//	kontroller.Din_Dout[0].kcc		:= 16#155;	// 01 - есть Целостность цепи для всех 5-ти выходов (в ЭЛПК-03-02 нет целостности выходов) 		
	K_Din_Dout_kk.kcc	:=	16#155;		// 01 - есть Целостность цепи для всех 5-ти выходов (в ЭЛПК-03-02 нет целостности выходов !!!)

//	kontroller.Din_Dout[0].value_cc	:= kontroller.Dout_[0];	//	содержимое выходных регистров		
	K_Din_Dout_kk.value_cc	:=	K_Dout;	//	содержимое выходных регистров

	// 01 - пассивное состояние			 10 - активное состояние 		
	K_Din_Dout_kk.kk.0	:=	NOT K_Dout.0;
	K_Din_Dout_kk.kk.1	:=	    K_Dout.0;
	// 01 - пассивное состояние			 10 - активное состояние 		
	K_Din_Dout_kk.kk.2	:=	NOT K_Dout.1;
	K_Din_Dout_kk.kk.3	:=	    K_Dout.1;
	// 01 - пассивное состояние			 10 - активное состояние 		
	K_Din_Dout_kk.kk.4	:=	NOT K_Dout.2;
	K_Din_Dout_kk.kk.5	:=	    K_Dout.2;
	// 01 - пассивное состояние			 10 - активное состояние 		
	K_Din_Dout_kk.kk.6	:=	NOT K_Dout.3;
	K_Din_Dout_kk.kk.7	:=	    K_Dout.3;
	// 01 - пассивное состояние			 10 - активное состояние 		
	K_Din_Dout_kk.kk.8	:=	NOT K_Dout.4;
	K_Din_Dout_kk.kk.9	:=	    K_Dout.4;

	// 01 - пассивное состояние			 10 - активное состояние 		
	K_Din_Dout_kk.kk.10	:=	NOT K_Dout.5;
	K_Din_Dout_kk.kk.11	:=	    K_Dout.5;
	// 01 - пассивное состояние			 10 - активное состояние 		
	K_Din_Dout_kk.kk.12	:=	NOT K_Dout.6;
	K_Din_Dout_kk.kk.13	:=	    K_Dout.6;
	// 01 - пассивное состояние			 10 - активное состояние 		
	K_Din_Dout_kk.kk.14	:=	NOT K_Dout.7;
	K_Din_Dout_kk.kk.15	:=	    K_Dout.7;

END_FUNCTION

// K2/std12k5/MAIN
PROGRAM MAIN
VAR

END_VAR


ELPK03_to_MLP_IN();// читать входы ЭЛПК-03-02 и передать в массивы 04

MainUP_PRG();// диагностика и OPC


///////////////////////////////////////////////////////////////////////////////////////////////////////////////////////
callExec(kontrollers);

{IF defined(imit)}
	{warning 'РЕЖИМ ИМИТАЦИИ! Входы и выходы отключены от физического источника'}
{ELSE}
execKontrollersInputs(table:=kontrollers);
{END_IF}

//SIP ();
callExec (YstTable);
callExec(imTable);
ProtectManager ();
OPC_Imit ();
algManager();
PPU_Init_ ();
Off_Q ();
{IF NOT defined(imit)}
execKontrollersOutputs(table:=kontrollers);
{END_IF}
///////////////////////////////////////////////////////////////////////////////////////////////////////////////////////

ELPK03_to_MLP_OUT(DO2_BLK:= 16#FF00, DO3_BLK:= 16#18FF);	// читать массивы 04 и передать в выходы ЭЛПК-03-02
										// с блокировкой ст байта DO_K[2] для индикации резервирования
										// с блокировкой мл байта DO_K[3] (сигналы резервирования старого) + DO_K[3].11 + DO_K[3].12 (индикация активности К1 и К2)

END_PROGRAM

// LowLevel_Algoritms/algoritms/Rassoglasovanie_dPmg
{attribute 'symbol' := 'none'}
FUNCTION_BLOCK PUBLIC Rassoglasovanie_dPmg EXTENDS BaseIM
VAR_INPUT
	di:REFERENCE TO singleSignal;
	ai:REFERENCE TO AISource;
END_VAR
VAR_OUTPUT
END_VAR
VAR
END_VAR

SUPER^();
IF	((di.q) AND (ai.value >= (ai.LA + 10))) OR ((NOT di.q) AND (ai.value <= (ai.LA - 10))) THEN
	statusSet.setBit (bitNum:=0,value:=1);
ELSE
	statusSet.setBit (bitNum:=0,value:=0);
END_IF

END_FUNCTION_BLOCK

// lowLevel_ecl/im/BaseIms/BaseIm
	{attribute 'symbol' := 'none'}
FUNCTION_BLOCK BaseIm EXTENDS BaseObject
IMPLEMENTS ObjectCommands, IImArchObject
VAR_INPUT
		{attribute 'symbol' := 'readwrite'}
	command:WORD;
END_VAR
VAR

END_VAR
VAR_OUTPUT
	{attribute 'symbol' := 'read'}
	status:DWORD;
	CommandFault:BOOL;
END_VAR
VAR
	statusSet:smartPack:=(status:=status);	
	objectTable:TableDescriptor;
	
	_command:WORD:=0;
	_haveCommand:BOOL;
	_logTwoCommands:AloneLogMessage;
	_cmd:UINT;
	_source:UINT;
	_error:UINT;
	_errorReset:TON:=(PT:=T#15S);
	_cmdReset:TON:=	(PT:=T#1S);
	_needResetCmd:BOOL;
	_opcCommandsDisabled:BOOL:=FALSE;
END_VAR

processObjectTable();

SUPER^();
_haveCommand:=FALSE;

statusSet.reset();

_errorReset(IN:=(_error<>0));

_command:=command;
command:=0;

IF _errorReset.Q THEN
	_error:=0;
	writeCommandToStatus();
END_IF

_cmdReset();
IF _needResetCmd AND _cmdReset.Q THEN
	resetCommand();
END_IF

IF hasCommand THEN
	onCommandActive(command:=_cmd);
END_IF

CommandFault:=_error<>0;

statusSet.setBit(21,_opcCommandsDisabled);

PROPERTY archName : STRING
GET
archName:=name;
END_GET
END_PROPERTY

PROPERTY archStatus : DWORD
GET
archStatus:=status;
END_GET
END_PROPERTY

METHOD PUBLIC DisableOpcControl
VAR_INPUT
END_VAR
VAR
	curObject:POINTER TO BaseObject;
	IcurIm:ObjectCommands;
END_VAR
_opcCommandsDisabled:=TRUE;

curObject:=objectTable.head;
IF curObject<>0 THEN
	REPEAT
		IF (__QUERYINTERFACE(curObject^,IcurIm)) THEN		
			IcurIm.DisableOpcControl();
		END_IF;
		curObject:=curObject^.getNext();
	UNTIL curObject=0
	END_REPEAT;
END_IF;
END_METHOD

METHOD EnableOpcControl
VAR_INPUT

END_VAR
VAR
	curObject:POINTER TO BaseObject;
	IcurIm:ObjectCommands;
END_VAR
_opcCommandsDisabled:=FALSE;

curObject:=objectTable.head;
IF curObject<>0 THEN
	REPEAT
		IF (__QUERYINTERFACE(curObject^,IcurIm)) THEN		
			IcurIm.EnableOpcControl();
		END_IF;
		curObject:=curObject^.getNext();
	UNTIL curObject=0
	END_REPEAT;
END_IF;
END_METHOD

METHOD FINAL execCommand
VAR_INPUT
END_VAR
VAR
	comUnp: SmartUnpack;
END_VAR
IF NOT _opcCommandsDisabled THEN
	IF _command<>0 THEN
		comUnp(value:=_command);	
		_source:=comUnp.getBits(13,15);
		IF _source<>0 THEN
			processCmd(cmd:=comUnp.getBits(0,2),sender:=_source,parametr:=comUnp.getBits(3,12));
		END_IF;
	END_IF;
END_IF;

ExecComands(objectTable);
END_METHOD

PROPERTY hasCommand : BOOL
GET
hasCommand:=(NOT _needResetCmd) AND (_cmd<>0);
END_GET
END_PROPERTY

PROPERTY PUBLIC opcCommandsDisabled : bool
GET
opcCommandsDisabled:=_opcCommandsDisabled;
END_GET
END_PROPERTY

METHOD PRIVATE writeCommandToStatus
VAR_INPUT
END_VAR
statusSet.setBits(23,25,_error);
statusSet.setBits(26,28,_cmd);
statusSet.setBits(29,31,_source);
END_METHOD

METHOD PROTECTED processObjectTable
VAR_INPUT
END_VAR
callExec(table:=objectTable);
END_METHOD

METHOD PROTECTED checkCmd : BOOL
VAR_INPUT
END_VAR
VAR
	
END_VAR
checkCmd:=_haveCommand;
IF _haveCommand THEN
	_logTwoCommands.write(CmpLog.LogClass.LOG_WARNING,name,'Two commands: ');
END_IF
_haveCommand:=TRUE;
END_METHOD

METHOD PROTECTED resetCommand
VAR_INPUT
END_VAR
IF _cmdReset.Q THEN
	_cmd:=0;
	_source:=0;
	writeCommandToStatus();
	_cmdReset(IN:=FALSE);
	_needResetCmd:=FALSE;
ELSE
	_needResetCmd:=TRUE;
END_IF;
END_METHOD

METHOD PROTECTED errorCommand
VAR_INPUT
END_VAR
_error:=_cmd;
resetCommand();
END_METHOD

//Метод вызывается каждый такт пересчета пока идет выполенение команды.
METHOD PROTECTED onCommandActive
VAR_INPUT
	command:WORD;
END_VAR
errorCommand();
END_METHOD

METHOD PROTECTED processCmd;
VAR_INPUT
	cmd:UINT;
	sender:UINT;
	parametr:UINT;
END_VAR
END_METHOD

METHOD PROTECTED setCmd
VAR_INPUT
	nCmd:uint;
END_VAR
checkCmd();
_cmd:=nCmd;
_error:=0;

_cmdReset(in:=FALSE);
_cmdReset.IN:=TRUE;	
	
_needResetCmd:=FALSE;
writeCommandToStatus();
END_METHOD

METHOD PUBLIC sendCommand
VAR_INPUT
	source:cmdSources;
	parametr:UINT;
	cmd:UINT;
END_VAR
_command:= SHL(source AND 16#7,13) OR SHL(parametr AND 16#3FF ,3) OR (cmd AND 16#3);
execCommand();
END_METHOD

METHOD PUBLIC writeImStatus
VAR_INPUT
END_VAR
END_METHOD

METHOD PUBLIC CommandFail : bool
VAR_INPUT
END_VAR
CommandFail:=_error<>0;
END_METHOD

END_FUNCTION_BLOCK

// lowLevel_ecl/Common/smartPack/smartPack
	{attribute 'symbol' := 'none'}
	{attribute 'reflection'}
FUNCTION_BLOCK smartPack//Упаковывает биты в двойное слово. 
(*Выдает ошибку в журнал если полсе reset() записывались одни и теже биты.
*)
VAR_INPUT	
	status:REFERENCE TO DWORD;//указатель на двойное слово
END_VAR
VAR_OUTPUT
END_VAR
VAR
	settedBits:DWORD;
	bitsAlredySetted:AloneLogMessage;
	bitsOutOfRenge:AloneLogMessage;
	{attribute 'instance-path'} 
	{attribute 'noinit'} 
	name: STRING; 
END_VAR
VAR CONSTANT

END_VAR

METHOD PUBLIC reset //сброс контроля перезаписи
VAR_INPUT
END_VAR
settedBits:=0;
END_METHOD

METHOD setBit 
//установить 1 бит
VAR_INPUT
	bitNum:WORD;// номер бита (с 0)
	value:BOOL;//Значение бита
END_VAR
setBits(bitNum,bitNum,bool_to_word(value));
END_METHOD

METHOD PUBLIC setBits //Устанавливает последовательность бит
VAR_INPUT
	start:WORD;//номер первого бита(с 0) 
	end:WORD;//номер последнего бита(с 0)
	value:DWORD;//значение. Записывается start-end+1 младших бит.
END_VAR
VAR
	statusMask:DWORD;
	bitsCount:WORD;
END_VAR
IF (start<0) OR (start>31) OR (end<0) OR (end>31) OR (start>end) THEN
	bitsOutOfRenge.write(CmpLog.LogClass.LOG_ERROR,name,'Nums out of range: ');	
	RETURN;
END_IF

bitsCount:=end-start+1;
statusMask:=SHL(SHL(1,bitsCount)-1,start);
IF (settedBits AND statusMask)<>0 THEN
	bitsAlredySetted.write(CmpLog.LogClass.LOG_ERROR,name,'Conflict bits: ');
END_IF
settedBits:=settedBits OR statusMask;
status:=(status AND NOT statusMask) OR (SHL(value,start) AND statusMask);
END_METHOD

END_FUNCTION_BLOCK

// lowLevel_ecl/Common/smartPack/SmartUnpack
{attribute 'symbol' := 'none'}
FUNCTION_BLOCK SmartUnpack//Распаковывает слово
VAR_INPUT
	value:WORD; //Значение
END_VAR
VAR_OUTPUT
END_VAR
VAR
END_VAR

METHOD getBit : BOOL
VAR_INPUT
	start:WORD;
END_VAR
getBit:= getBits(start,start)<>0;
END_METHOD

METHOD getBits : Word
VAR_INPUT
	start:WORD;
	end: WORD;
END_VAR
VAR
	statusMask:WORD;
	bitsCount:WORD;
END_VAR
bitsCount:=end-start+1;
statusMask:=SHL(SHL(1,bitsCount)-1,start);
getBits:=SHR(value AND statusMask,start);
END_METHOD

END_FUNCTION_BLOCK

// lowLevel_ecl/im/BaseIms/singleSignal
{attribute 'symbol' := 'none'}
FUNCTION_BLOCK singleSignal EXTENDS BaseIm
VAR_INPUT
	signal:REFERENCE TO ReliableBit;
END_VAR
VAR_OUTPUT
	Q:BOOL;
	reliability:BOOL;
END_VAR
VAR
END_VAR

SUPER^();
IF __ISVALIDREF(signal) THEN
	Q:=checkArg(signal);
	reliability:=signal.reliability;
END_IF

METHOD PUBLIC writeImStatus
VAR_INPUT
END_VAR
SUPER^.writeImStatus();
statusSet.setBit(0,Q);
END_METHOD

END_FUNCTION_BLOCK

// lowLevel_ecl/Common/functions/checkArg
FUNCTION checkArg : BOOL
VAR_INPUT
	chBit:REFERENCE TO ReliableBit;
END_VAR
VAR
END_VAR

checkArg:=FALSE;
IF __ISVALIDREF(chBit) THEN
	IF chBit.reliability THEN
		checkArg:=chBit.value;
	END_IF
END_IF

END_FUNCTION

// lowLevel_ecl/kontroller/baseSources/ReliableBit
	{attribute 'symbol' := 'none'}
FUNCTION_BLOCK ReliableBit
VAR_INPUT
END_VAR
VAR_OUTPUT
	value:BOOL;//Значение	
	reliability:BOOL;//достоверный
END_VAR
VAR
	
END_VAR

PROPERTY PUBLIC ReliableFalse : Bool
GET
ReliableFalse:= (NOT value) AND reliability;
END_GET
END_PROPERTY

PROPERTY PUBLIC ReliableTrue : Bool
GET
ReliableTrue:=value AND reliability;
END_GET
END_PROPERTY

METHOD setReliability
VAR_INPUT
	rel:BOOL;
END_VAR
reliability:=rel;
END_METHOD

METHOD PUBLIC setValue
VAR_INPUT
	val: BOOL;
END_VAR
value:=val;
END_METHOD

END_FUNCTION_BLOCK

// lowLevel_ecl/kontroller/baseSources/AISource
	{attribute 'symbol' := 'none'}
FUNCTION_BLOCK AISource EXTENDS BaseIm
IMPLEMENTS ISource, IAnalogArchObject, IAiSource
VAR_INPUT
	addr:WORD;
	
	dLL:REAL:=RNaN(); 
	dHL:REAL:=RNaN(); 
	dLA:REAL:=RNaN();
	dHA:REAL:=RNaN();
	dLW:REAL:=RNaN();
	dHW:REAL:=RNaN();  
	dmaxChangeSpeed:REAL:=RNaN();  
END_VAR
VAR_OUTPUT
		{attribute 'symbol' := 'readwrite'}
	value:REAL;

	interval:statusAi;
	
	remont	:	BOOL	;	//	bit-0 вывод канала в ремонт  1-есть, 0 –нет				
	{attribute 'symbol' := 'read'} 
	LL	:	REAL	:=RNaN();	//	Нижняя граница физического диапазона	Для преобразования из 4-20 мА и отображения в SCADA.
	{attribute 'symbol' := 'read'} 
	HL	:	REAL	:=RNaN();	//	Верхняя граница физического диапазона	Для преобразования из 4-20 мА и отображения в SCADA.
	{attribute 'symbol' := 'read'} 
	HA	:	REAL	:=RNaN();	//	Верхняя аварийная граница	Уставка срабатывания аварийного останова по повышению параметра
	{attribute 'symbol' := 'read'} 
	HW	:	REAL	:=RNaN();	//	Верхняя предупредительная граница	Уставка срабатывания предупредительной сигнализации по повышению параметра
	{attribute 'symbol' := 'read'} 
	LW	:	REAL	:=RNaN();	//	Нижняя предупредительная граница	Уставка срабатывания предупредительной сигнализации по понижению параметра
	{attribute 'symbol' := 'read'} 
	LA	:	REAL	:=RNaN();	//	Верхняя аварийная граница	Уставка срабатывания аварийного останова по понижению параметра
	{attribute 'symbol' := 'read'} 
	histeresis	:	REAL	;	//	Гистерезис.( % от физической шкалы) Уставка устранения дребезга по предупредительной сигнализации	Для устранения частого срабатывания предупредительной сигнализации при колебания около границы	
	//_de	:	REAL	;	//	Уставка рассогласования от аппаратных границ	Разница тока для формирования неисправности канала по выходу за диапазон измерения.
	{attribute 'symbol' := 'read'} 
	aperturFilter	:	REAL	;	//	Уставка апертурного фильтра	При применении апертурного фильтра, фильтрация малых изменений сигнала
	{attribute 'symbol' := 'read'} 
	pikFiler	:	REAL	;	//	Уставка пикового фильтра	При применении пикового фильтра, фильтрация пиков, случайных бросков сигнала
	{attribute 'symbol' := 'read'} 
	exponentialFilter	:	REAL	:=RNaN();	//	Уставка экпоненциального фильтра	При применении экспоненциального фильтра.
	{attribute 'symbol' := 'read'}
	rassoglasovanie	:	REAL	;	//	Уставка рассогласования от аппаратных границ. В процентах от диапазона.
	{attribute 'symbol' := 'read'}	
	maxChangeSpeed:REAL; //Максимальная скорость изменения сигнала 1/сек
	{attribute 'symbol' := 'read'} 
	ChangeSpeed:REAL;//Скорость изменения.
END_VAR
VAR
	{attribute 'symbol' := 'readwrite'}
	newLL:REAL;  // новые границы
	{attribute 'symbol' := 'readwrite'}
	newHL:REAL;  // новые границы
	{attribute 'symbol' := 'readwrite'}
	newLA:REAL;  // новые границы
	{attribute 'symbol' := 'readwrite'}
	newHA:REAL;  // новые границы
	{attribute 'symbol' := 'readwrite'}
	newLW:REAL;  // новые границы
	{attribute 'symbol' := 'readwrite'}
	newHW:REAL;  // новые границы		

	_imit:BOOL;  
	_notReliable:BOOL;
	_disabledAlarms:BYTE;
	
	_lastValue:REAL:=RNaN();
	_LastValueTimer:TON:=(PT:=T#1S);
	_normalTrig:R_TRIG;
END_VAR

VAR CONSTANT
	cmd_SetUstavki:WORD:=1;
	cmd_SetRemont:WORD:=2;
	cmd_ResetRemont:WORD:=3;
	cmd_kvitNotReliable:WORD:=4;
END_VAR
VAR_TEMP
	srcInterval:statusAi;
END_VAR

SUPER^();

IF NOT imit THEN
	value:=getData(o_interval=>srcInterval);
	
	value:=apFilter(value,_lastValue);
	value:=exponential(value,_lastValue);
ELSE
	srcInterval:=statusAi.normal;
END_IF;

IF NOT notReliable THEN
	IF srcInterval=statusAi.normal THEN
		interval:=CalkLimits();
	ELSE
		interval:=srcInterval;
	END_IF;
ELSE
	interval:=statusAi.NOTRELIABLE;
END_IF	

IF remont THEN
	interval:=statusAi.NOTDEFINED;
END_IF


_normalTrig(CLK:=interval>=statusAi.normal);

IF (NOT FPU.IsRealNaN(_lastValue)) AND (NOT _normalTrig.Q) THEN
	_LastValueTimer();
	IF (value<>_lastValue) OR _LastValueTimer.Q THEN
		IF (_LastValueTimer.ET>T#0MS) THEN
			ChangeSpeed:=(value-_lastValue)/(TIME_TO_REAL(_LastValueTimer.ET)/1000);
		END_IF
		_LastValueTimer(IN:=FALSE);
		_LastValueTimer(IN:=TRUE);
	END_IF
END_IF

_lastValue:=value;

IF (NOT FPU.IsRealNaN(maxChangeSpeed)) AND (maxChangeSpeed>0) THEN
	IF (interval>=statusAi.normal) THEN		
		IF ABS(ChangeSpeed)>maxChangeSpeed THEN
			 notReliable:=TRUE;
		END_IF
	END_IF
END_IF

PROPERTY aiInterval : statusAi
GET
aiInterval:=interval;
END_GET
END_PROPERTY

PROPERTY aiRemont : BOOL
GET
aiRemont:=remont;
END_GET
END_PROPERTY

PROPERTY aiValue : REAL
GET
aiValue:=value;
END_GET
END_PROPERTY

METHOD PRIVATE apFilter: REAL
VAR_INPUT
	currentValue:REAL;
	lastValue:REAL;
END_VAR
VAR
	ap:REAL;
END_VAR
IF NOT FPU.IsRealNaN(aperturFilter) THEN
	ap:=aperturFilter*0.01*(Hl-Ll);
	IF rABS(currentValue-lastValue)>ap THEN
		apFilter:=currentValue;
	ELSE
		apFilter:=lastValue;
	END_IF
ELSE
	apFilter:=currentValue;
END_IF
END_METHOD

PROPERTY archName : STRING
GET
END_GET
END_PROPERTY

PROPERTY archSrcValue : REAL
GET
END_GET
END_PROPERTY

PROPERTY archStatus : DWORD
GET
END_GET
END_PROPERTY

PROPERTY archValue : REAL
GET
archValue:=value;
END_GET
END_PROPERTY

METHOD PROTECTED CalkLimits:statusAi
VAR_INPUT

END_VAR
VAR
	h:REAL:=0;
	mismatch:REAL:=0;
END_VAR
CalkLimits:=statusAi.NOTDEFINED;

IF NOT (FPU.IsRealNaN(ll) OR FPU.IsRealNaN(Hl))THEN
	h := histeresis* 0.01 * (Hl-Ll);
	mismatch:=rassoglasovanie* 0.01 * (Hl-Ll);
	
	IF ( value < LL-mismatch)   THEN
		CalkLimits:=statusAi.LL;
		RETURN;
	END_IF  
	IF  (value > Hl+mismatch) THEN
		CalkLimits:=statusAi.HL;
		RETURN;
	END_IF
END_IF

IF (NOT FPU.IsRealNaN(la)) AND ((disabledAlarms AND AnalogAlarms.LA)=0) THEN
	IF (value  < La) OR ((interval=statusAi.LA)  AND ( (value -h) < La))  THEN 
		CalkLimits:=statusAi.LA;
		RETURN;
	END_IF
END_IF 

IF NOT FPU.IsRealNaN(Ha) AND ((disabledAlarms AND AnalogAlarms.HA)=0)THEN
	IF (value > Ha) OR ((interval=statusAi.HA)  AND ( (value +h) > HA))  THEN 
		CalkLimits:=statusAi.HA;
		RETURN;
	END_IF
END_IF

IF NOT FPU.IsRealNaN(LW) AND ((disabledAlarms AND AnalogAlarms.LW)=0) THEN
	IF (value < LW) OR ((interval=statusAi.LW)  AND ( (value -h) < Lw))   THEN 
		CalkLimits:=statusAi.LW;
		RETURN;
	END_IF
END_IF

IF NOT FPU.IsRealNaN(HW) AND ((disabledAlarms AND AnalogAlarms.HW)=0)THEN
	IF (value  > HW)  OR ((interval=statusAi.HW)  AND ( (value +h) > Hw))   THEN 
		CalkLimits:=statusAi.HW;
		RETURN;
	END_IF
END_IF

CalkLimits:=statusAi.normal;
END_METHOD

{attribute 'symbol' := 'none'}
PROPERTY PUBLIC disabledAlarms : BYTE
GET
disabledAlarms:=_disabledAlarms;
END_GET
SET
_disabledAlarms:=disabledAlarms;
END_SET
END_PROPERTY

METHOD PRIVATE exponential : Real
VAR_INPUT
	currentValue:REAL;
	lastValue:REAL;
END_VAR
IF (NOT FPU.IsRealNaN(exponentialFilter)) AND (exponentialFilter<>0) AND (NOT FPU.IsRealNaN(lastValue)) THEN
	exponential:=exponentialFilter*currentValue+(1-exponentialFilter)*lastValue;
ELSE
	exponential:=currentValue;
END_IF
END_METHOD

METHOD PROTECTED GetData : Real
VAR_INPUT
END_VAR
VAR_OUTPUT
	o_interval:statusAi;
END_VAR
END_METHOD

{attribute 'symbol' := 'none'}
PROPERTY imit : BOOL
GET
imit:=_imit;
END_GET
SET
_imit:=imit;
END_SET
END_PROPERTY

METHOD kvitNotReliable
VAR_INPUT
END_VAR
setCmd(nCmd:=cmd_kvitNotReliable);

_notReliable:=FALSE;

resetCommand();
END_METHOD

{attribute 'symbol' := 'none'}
PROPERTY PUBLIC notReliable : bool
GET
notReliable:=_notReliable;
END_GET
SET
IF notReliable THEN
	_notReliable:=notReliable;
	interval:=statusAi.NOTRELIABLE;
END_IF
END_SET
END_PROPERTY

METHOD PROTECTED processCmd;
VAR_INPUT
	cmd:UINT;
	sender:UINT;
	parametr:UINT;
END_VAR
CASE cmd OF
	cmd_SetUstavki:setUstavki(nLL:=newLL,nLA:=newLA, nLW:=newLW, nHW:=newHW, nHa:=newHA,nHl:=newHL,flags:= parametr);
	cmd_SetRemont:setRemont();
	cmd_ResetRemont:resetRemont();
	cmd_kvitNotReliable:kvitNotReliable();
END_CASE
END_METHOD

METHOD PROTECTED readPersistent
VAR_INPUT
END_VAR
Ll:=FPU.StrToReal(readValue());
la:=FPU.StrToReal(readValue());
lw:=FPU.StrToReal(readValue());
hw:=FPU.StrToReal(readValue());
ha:=FPU.StrToReal(readValue());
Hl:=FPU.StrToReal(readValue());
remont:=STRING_TO_BOOL(readValue());
histeresis:=FPU.StrToReal(readValue());
aperturFilter:=FPU.StrToReal(readValue());
pikFiler:=FPU.StrToReal(readValue());
exponentialFilter:=FPU.StrToReal(readValue());
rassoglasovanie:=FPU.StrToReal(readValue());
maxChangeSpeed:=FPU.StrToReal(readValue());
END_METHOD

METHOD resetRemont
VAR_INPUT
END_VAR
setCmd(nCmd:=cmd_ResetRemont);

remont:=FALSE;

SaveToFile();

resetCommand();
END_METHOD

METHOD PROTECTED setDefaultPersistent:BOOL
VAR_INPUT
END_VAR
LL:=dLL;
LA:=dLA;
LW:=dLW;
HW:=dHW;
Ha:=dHA;
Hl:=dHL;
maxChangeSpeed:=dmaxChangeSpeed;
setDefaultPersistent:=TRUE;
END_METHOD

METHOD setRemont
VAR_INPUT
END_VAR
setCmd(nCmd:=cmd_SetRemont);

remont:=TRUE;

SaveToFile();

resetCommand();
END_METHOD

METHOD setUstavki
VAR_INPUT
	nLL:REAL;
	nHl:REAL;
	nLA:REAL;
	nHa:REAL;
	nLW:REAL;
	nHW:REAL;
	flags:WORD:=16#FF;
END_VAR
setCmd(nCmd:=cmd_SetUstavki);

IF (flags AND AnalogLimitFlags.LL)<>0 THEN
	LL:=nLL;
END_IF
IF (flags AND AnalogLimitFlags.HL)<>0 THEN
	Hl:=nHl;
END_IF
IF (flags AND AnalogLimitFlags.LA)<>0 THEN
	LA:=nlA;
END_IF
IF (flags AND AnalogLimitFlags.HA)<>0 THEN
	Ha:=nha;
END_IF
IF (flags AND AnalogLimitFlags.LW)<>0 THEN
	LW:=nlW;
END_IF
IF (flags AND AnalogLimitFlags.HW)<>0 THEN
	HW:=nhw;
END_IF

SaveToFile();

resetCommand();
END_METHOD

METHOD PUBLIC writeImStatus
VAR_INPUT
END_VAR
VAR
	cInteval:statusAi;
END_VAR
SUPER^.writeImStatus();
statusSet.setBits(0,3,interval);
statusSet.setBit(4,remont);
statusSet.setBit(5,interval<statusAi.normal);
statusSet.setBits(6,9,_disabledAlarms);
END_METHOD

METHOD PROTECTED writePersistent
VAR_INPUT
END_VAR
writeValue(value:=FPU.RealToStr(Ll),comment:='LL');
writeValue(value:=FPU.RealToStr(la),comment:='LA');
writeValue(value:=FPU.RealToStr(lw),comment:='LW');
writeValue(value:=FPU.RealToStr(hw),comment:='HW');
writeValue(value:=FPU.RealToStr(ha),comment:='HA');
writeValue(value:=FPU.RealToStr(Hl),comment:='HL');
writeValue(value:=BOOL_TO_STRING(remont),comment:='Ремонт');
writeValue(value:=FPU.RealToStr(histeresis),comment:='Гистерезис');
writeValue(value:=FPU.RealToStr(aperturFilter),comment:='Апертурный фильтр');
writeValue(value:=FPU.RealToStr(pikFiler),comment:='Пиковый фильтр');
writeValue(value:=FPU.RealToStr(exponentialFilter),comment:='Экспоненциальный фильтр');
writeValue(value:=FPU.RealToStr(rassoglasovanie),comment:='Рассогласование');
writeValue(value:=FPU.RealToStr(maxChangeSpeed),comment:='Максимальная скорость изменения');
END_METHOD

END_FUNCTION_BLOCK

// lowLevel_ecl/kontroller/baseSources/IAiSource
INTERFACE IAiSource

PROPERTY aiInterval : statusAi
GET
END_GET
END_PROPERTY

PROPERTY aiRemont : BOOL
GET
END_GET
END_PROPERTY

PROPERTY aiValue : real
GET
END_GET
END_PROPERTY

END_INTERFACE

// lowLevel_ecl/Common/functions/RNaN
FUNCTION RNaN : real
VAR_INPUT
END_VAR
VAR
END_VAR

RNaN:=FPU.GetRealSpecialVal(fpu.ESpecial_FP_Value.NaN);

END_FUNCTION

// lowLevel_ecl/Common/functions/rABS
FUNCTION rABS : real
VAR_INPUT
	inp:REAL;
END_VAR
VAR
END_VAR

IF inp<0.0 THEN
	rABS:=-inp;
ELSE
	rABS:=inp;
END_IF

END_FUNCTION

// K1/std12k5/modbus/tstModbus
	{attribute 'symbol' := 'none'}
FUNCTION_BLOCK tstModbus EXTENDS MbKontroller
VAR_INPUT
END_VAR
VAR_OUTPUT
	di_1:DiSourceMb(table:=ADR(inputTable)):=(addr:=0);
	ai_1:AiSourceMb(table:=ADR(inputTable)):=(addr:=1,reliability:=di_1.bits[1]);
	ao_1:AoProxiMb(table:=ADR(outputTable)):=(addr:=5, source:=ai_1);
END_VAR
VAR
END_VAR

SUPER^();

METHOD PROTECTED ProcessInputs
VAR_INPUT
END_VAR
IF di_1.trigs[5].Qp THEN
	//команда
END_IF
END_METHOD

METHOD PROTECTED ProcessOutputs
VAR_INPUT
END_VAR
setOutputValue(addr:=5,1);
setOutputFloat(addr:=6,1.5);
END_METHOD

END_FUNCTION_BLOCK

// K2/std12k5/modbus/tstModbus
	{attribute 'symbol' := 'none'}
FUNCTION_BLOCK tstModbus EXTENDS MbKontroller
VAR_INPUT
END_VAR
VAR_OUTPUT
	di_1:DiSourceMb(table:=ADR(inputTable)):=(addr:=0);
	ai_1:AiSourceMb(table:=ADR(inputTable)):=(addr:=1,reliability:=di_1.bits[1]);
	ao_1:AoProxiMb(table:=ADR(outputTable)):=(addr:=5, source:=ai_1);
END_VAR
VAR
END_VAR

SUPER^();

METHOD PROTECTED ProcessInputs
VAR_INPUT
END_VAR
IF di_1.trigs[5].Qp THEN
	//команда
END_IF
END_METHOD

METHOD PROTECTED ProcessOutputs
VAR_INPUT
END_VAR
setOutputValue(addr:=5,1);
setOutputFloat(addr:=6,1.5);
END_METHOD

END_FUNCTION_BLOCK

// lowLevel_ecl/kontroller/modbus/MbKontroller
{attribute 'symbol' := 'none'}
FUNCTION_BLOCK MbKontroller EXTENDS baseKontroller
VAR_INPUT
	MbRole:MbKontrollerRole;
	slaveError:REFERENCE TO BOOL;
	slaveRestart:REFERENCE TO BOOL;
	restartDelay:TIME:=T#20S;
	restartDuration:TIME:=T#30S;
	AiWordOrder:MbAiWordOrder:=MbAiWordOrder.AiWordOrder12;
END_VAR
VAR_OUTPUT
	{attribute 'symbol' := 'read'}
	noLink:BOOL;
END_VAR
VAR
	input:ARRAY [1..500] OF WORD;
	holding:ARRAY [1..500] OF WORD;
	
	_init:BOOL;
	
	restartTimer:TON;
	noLinkTimer:TOF;
END_VAR

SUPER^();
IF NOT _init THEN
	setSourcesProp(table:=inputTable);
	setSourcesProp(table:=outputTable);
	_init:=TRUE;
END_IF
IF NOT imit THEN
	IF (__ISVALIDREF(slaveError)) THEN
		noLinkTimer(IN:=slaveError,PT:=restartDuration,Q=>noLink);
		IF (__ISVALIDREF(slaveRestart)) THEN
			restartTimer(IN:=slaveError AND (NOT slaveRestart),PT:=restartDelay,Q=>slaveRestart);
		END_IF
	END_IF
ELSE
	noLink:=FALSE;
END_IF

METHOD PUBLIC callInputTable
VAR_INPUT
END_VAR
SUPER^.callInputTable();
ProcessInputs();
END_METHOD

METHOD callOutputTable
VAR_INPUT
END_VAR
ProcessOutputs();
SUPER^.callOutputTable();
END_METHOD

METHOD PUBLIC getInputFloat : REAL
VAR_INPUT
	addr:WORD;
END_VAR
VAR
	rawValue:FloatAsWords;
END_VAR
CASE AiWordOrder OF
	MbAiWordOrder.AiWordOrder12:
		rawValue.wValue[0]:=getInputValue(addr:=addr);
		rawValue.wValue[1]:=getInputValue(addr:=addr+1);	
	MbAiWordOrder.AiWordOrder21:
		rawValue.wValue[0]:=getInputValue(addr:=addr+1);
		rawValue.wValue[1]:=getInputValue(addr:=addr);
END_CASE

getInputFloat:=rawValue.fValue;
END_METHOD

METHOD PUBLIC getInputValue : WORD
VAR_INPUT
	addr:WORD;
END_VAR
CASE MbRole OF
	MbKontrollerRole.MK_MASTER:
		getInputValue:=input[addr];
	MbKontrollerRole.MK_SLAVE:
		getInputValue:=holding[addr];
END_CASE
END_METHOD

METHOD PROTECTED ProcessInputs
VAR_INPUT
END_VAR
END_METHOD

METHOD PROTECTED ProcessOutputs
VAR_INPUT
END_VAR
END_METHOD

METHOD PUBLIC setOutputByte
VAR_INPUT
	addr:WORD;
	value:BYTE;
	usedByte:UsedByteMBSource;
END_VAR
VAR
	rawValue:FloatAsWords;
	
END_VAR


CASE MbRole OF
	MbKontrollerRole.MK_MASTER: 	
	rawValue.wValue[0]:=	holding[addr]; // сохраняем 
			IF usedByte=UsedByteMBSource.HB THEN 
				rawValue.bValue[1]:=	value;
			ELSE
				rawValue.bValue[0]:=	value;
			END_IF
		holding[addr]:=rawValue.wValue[0]; //кормим слово

	MbKontrollerRole.MK_SLAVE: 	
		rawValue.wValue[0]:=	input[addr]; // сохраняем 
			IF usedByte=UsedByteMBSource.HB THEN 
				rawValue.bValue[1]:=	value;
			ELSE
				rawValue.bValue[0]:=	value;
			END_IF
		input[addr]:=rawValue.wValue[0]; //кормим слово
END_CASE
END_METHOD

METHOD PUBLIC setOutputFloat
VAR_INPUT
	addr:WORD;
	value:REAL;
END_VAR
VAR
	rawValue:FloatAsWords;
END_VAR
rawValue.fValue:=value;
CASE AiWordOrder OF
	MbAiWordOrder.AiWordOrder12:
		setOutputValue(addr:=addr,value:=rawValue.wValue[0]);
		setOutputValue(addr:=addr+1,value:=rawValue.wValue[1]);	
	MbAiWordOrder.AiWordOrder21:
		setOutputValue(addr:=addr+1,value:=rawValue.wValue[0]);
		setOutputValue(addr:=addr,value:=rawValue.wValue[1]);	
END_CASE
END_METHOD

METHOD PUBLIC setOutputValue
VAR_INPUT
	addr:WORD;
	value:WORD;
END_VAR
CASE MbRole OF
	MbKontrollerRole.MK_MASTER:
		holding[addr]:=value;
	MbKontrollerRole.MK_SLAVE:
		input[addr]:=value;
END_CASE
END_METHOD

METHOD PRIVATE setSourcesProp
VAR_INPUT
	CONSTANT table:TableDescriptor;
END_VAR
VAR
	curObject:POINTER TO BaseObject;
	curSource:IMbSource;
END_VAR
curObject:=table.head;
IF curObject=0 THEN
	RETURN;
END_IF
REPEAT
	IF (__QUERYINTERFACE(curObject^,curSource)) THEN		
		curSource.setKontroller(THIS^);
	END_IF;
	curObject:=curObject^.getNext();
	UNTIL curObject=0
END_REPEAT
END_METHOD

END_FUNCTION_BLOCK

// lowLevel_ecl/kontroller/modbus/Sources/IMbSource
INTERFACE IMbSource EXTENDS __SYSTEM.IQueryInterface

METHOD setKontroller
VAR_INPUT
	nKontroller:REFERENCE TO MbKontroller;
END_VAR
END_METHOD

END_INTERFACE

// lowLevel_ecl/kontroller/modbus/Sources/DiSourceMb
{attribute 'symbol' := 'none'}
FUNCTION_BLOCK DiSourceMb EXTENDS DISource
IMPLEMENTS IMbSource;
VAR_INPUT
	
END_VAR
VAR_OUTPUT
	Trigs:array [0..15] OF RP_trig;
END_VAR
VAR
	mbKontr:REFERENCE TO MbKontroller;
	bitNumber:INT;
	I:INT;
END_VAR

SUPER^();

FOR I:=0 TO 15 DO
	IF bits[I].reliability THEN
  		Trigs[i](in:= bits[I].value);
	END_IF
END_FOR

METHOD PROTECTED getData : word
VAR_INPUT
END_VAR
VAR_OUTPUT
	reliability:WORD;
END_VAR
getData:=mbKontr.getInputValue(addr:=addr);
IF NOT mbKontr.noLink THEN
	reliability:=16#FFFF;
ELSE
	reliability:=16#0000;	
END_IF
END_METHOD

METHOD setKontroller
VAR_INPUT
	nKontroller	: REFERENCE TO MbKontroller;
END_VAR
mbKontr REF=nKontroller;
END_METHOD

END_FUNCTION_BLOCK

// lowLevel_ecl/kontroller/baseSources/DISource
	{attribute 'symbol' := 'none'}
FUNCTION_BLOCK DISource EXTENDS BaseObject
IMPLEMENTS ISource, IDiscretArchObject
VAR_INPUT
	addr:WORD;
END_VAR
VAR_OUTPUT
		bits:ARRAY [0..15] OF InversableReliableBit;
		{attribute 'symbol' := 'readwrite'}
		value:WORD;
		{attribute 'symbol' := 'readwrite'}
		reliability:WORD;
END_VAR
VAR
	_imit:BOOL;  
END_VAR
VAR_TEMP
	bitNumber:INT;
END_VAR

SUPER^();
IF NOT imit THEN
	value:=getData(reliability=>reliability);
END_IF;

FOR bitNumber:=0 TO 15 DO
	bits[bitNumber].setReliability(UINT_TO_BOOL(SHR (reliability, bitNumber) AND 16#1));
	IF bits[bitNumber].reliability THEN
		bits[bitNumber].setValue(UINT_TO_BOOL(SHR (value, bitNumber) AND 16#1));
	END_IF;
END_FOR

PROPERTY archName : STRING
GET
archName:=name;
END_GET
END_PROPERTY

PROPERTY archReliability : WORD
GET
archReliability:=reliability;
END_GET
END_PROPERTY

PROPERTY archValue : WORD
GET
archValue:=value;
END_GET
END_PROPERTY

METHOD PROTECTED getData : word
VAR_INPUT
END_VAR
VAR_OUTPUT
	reliability:WORD;
END_VAR
END_METHOD

{attribute 'symbol' := 'none'}
PROPERTY imit : BOOL
GET
imit:=_imit;
END_GET
SET
_imit:=imit;
END_SET
END_PROPERTY

END_FUNCTION_BLOCK

// lowLevel_ecl/kontroller/baseSources/InversableReliableBit
	{attribute 'symbol' := 'none'}
FUNCTION_BLOCK InversableReliableBit EXTENDS ReliableBit
VAR_INPUT
END_VAR
VAR_OUTPUT

END_VAR
VAR
	_inversed:ReliableBit;
END_VAR

{attribute 'symbol' := 'none'}
PROPERTY inverse : REFERENCE TO ReliableBit;
GET
inverse ref=_inversed;
END_GET
END_PROPERTY

METHOD setReliability
VAR_INPUT
	rel:BOOL;
END_VAR
SUPER^.setReliability(rel);
_inversed.setReliability(rel);
END_METHOD

METHOD PUBLIC setValue
VAR_INPUT
	val: BOOL;
END_VAR
SUPER^.setValue(val);
_inversed.setValue(NOT val);
END_METHOD

END_FUNCTION_BLOCK

// lowLevel_ecl/kontroller/modbus/Sources/AiSourceMb
{attribute 'symbol' := 'none'}
FUNCTION_BLOCK AiSourceMb EXTENDS AISource
IMPLEMENTS IMbSource;
VAR_INPUT
	k:REAL:=1;
	b:REAL:=0;
	reliability:REFERENCE TO ReliableBit;
	extInterval:REFERENCE TO DISource;
END_VAR
VAR_OUTPUT
END_VAR
VAR
	mbKontr:REFERENCE TO MbKontroller;
	source:AnalogRecalc;
END_VAR

SUPER^();

METHOD PROTECTED GetData : Real
VAR_INPUT
END_VAR
VAR_OUTPUT
	o_interval:statusAi;
END_VAR
VAR
	intervalUnp:SmartUnpack;
END_VAR
source.input:=mbKontr.getInputFloat(addr:=addr);
source.k:=k;
source.b:=b;
source.h:=histeresis;
source.ap:=aperturFilter;
source.dp:=pikFiler;
source.ds:=exponentialFilter;
source.de:=rassoglasovanie;
source();

GetData:=source.value;

IF (mbKontr.noLink) AND NOT _imit THEN
	o_interval:=statusAi.NOTDEFINED;
ELSE
	IF (__ISVALIDREF(extInterval)) THEN
		intervalUnp.value:=extInterval.value;
		o_interval:=WORD_TO_BYTE(intervalUnp.getBits(0,3));
	ELSE
		IF __ISVALIDREF(reliability) THEN
			IF reliability.reliability AND reliability.value THEN
				o_interval:=statusAi.normal;
			ELSE
				o_interval:=statusAi.NOTDEFINED;
			END_IF
		ELSE
			o_interval:=statusAi.normal;	
		END_IF
	END_IF
END_IF
END_METHOD

METHOD setKontroller
VAR_INPUT
	nKontroller	: REFERENCE TO MbKontroller;
END_VAR
mbKontr REF=nKontroller;
END_METHOD

END_FUNCTION_BLOCK

// lowLevel_ecl/Common/fb/AnalogRecalc
	{attribute 'symbol' := 'none'}
FUNCTION_BLOCK AnalogRecalc
VAR_INPUT		
	k:REAL;
	b:REAL;
	input:REAL;//входное значение
	
	h	:	REAL	;	//	Гистерезис.( % от физической шкалы) Уставка устранения дребезга по предупредительной сигнализации	Для устранения частого срабатывания предупредительной сигнализации при колебания около границы
	ap	:	REAL	;	//	Уставка апертурного фильтра	При применении апертурного фильтра, фильтрация малых изменений сигнала 
	dp	:	REAL	;	//	Уставка пикового фильтра	При применении пикового фильтра, фильтрация пиков, случайных бросков сигнала 
	ds	:	REAL	;	//	Уставка экпоненциального фильтра	При применении экспоненциального фильтра.

	de	:	REAL	;	//	Уставка рассогласования от аппаратных границ	Разница тока для формирования неисправности канала по выходу за диапазон измерения.
END_VAR
VAR_OUTPUT
	value:REAL;
END_VAR
VAR
END_VAR
VAR_TEMP
END_VAR

	value := k*input +b;

END_FUNCTION_BLOCK

// lowLevel_ecl/kontroller/modbus/Sources/AoProxiMb
{attribute 'symbol' := 'none'}
FUNCTION_BLOCK PUBLIC AoProxiMb EXTENDS AOSource
IMPLEMENTS IMbSource;
VAR_INPUT
	k:REAL:=1;
	b:REAL:=0;
	Source:REFERENCE TO AISource;
END_VAR
VAR_OUTPUT
END_VAR
VAR
	mbKontr:REFERENCE TO MbKontroller;
END_VAR

SUPER^();

METHOD setKontroller
VAR_INPUT
	nKontroller: REFERENCE TO MbKontroller;
END_VAR
mbKontr REF=nKontroller;
END_METHOD

METHOD PROTECTED writeData
VAR_INPUT
	val:REAL;
END_VAR
VAR
	rawValue:FloatAsWords;	
END_VAR
IF __ISVALIDREF(Source) THEN
	rawValue.fValue:=Source.value;
	mbKontr.setOutputValue(addr:=addr+2,value:=Source.interval);
ELSE
	rawValue.fValue:=k*val+b;	
END_IF

mbKontr.setOutputFloat(addr:=addr,value:=rawValue.fValue);
END_METHOD

END_FUNCTION_BLOCK

// lowLevel_ecl/kontroller/baseSources/AOSource
	{attribute 'symbol' := 'none'}
FUNCTION_BLOCK AOSource EXTENDS BaseIm
IMPLEMENTS ISource, IAnalogArchObject
VAR_INPUT
	addr:WORD;
	
		{attribute 'symbol' := 'readwrite'}
	newLL	:	REAL	;	//	Нижняя граница физического диапазона	Для преобразования из 4-20 мА и отображения в SCADA.
		{attribute 'symbol' := 'readwrite'}
	newHL	:	REAL	;	//	Верхняя граница физического диапазона	Для преобразования из 4-20 мА и отображения в SCADA.
	
	dLL:REAL:=RNaN(); 
	dHL:REAL:=RNaN(); 
END_VAR
VAR_OUTPUT
		{attribute 'symbol' := 'read'}
	Value:REAL;
	
		{attribute 'symbol' := 'read'}
	LL	:	REAL	;	//	Нижняя граница физического диапазона	Для преобразования из 4-20 мА и отображения в SCADA.
	{attribute 'symbol' := 'read'}
	HL	:	REAL	;	//	Верхняя граница физического диапазона	Для преобразования из 4-20 мА и отображения в SCADA.	
END_VAR
VAR
		{attribute 'symbol' := 'readwrite'}
	newValue:REAL;

	_imit:BOOL;  
END_VAR

VAR CONSTANT
	cmd_ChangeValue:WORD:=1;
	cmd_ChangeLimits:WORD:=2;
END_VAR

SUPER^();
IF NOT imit THEN
	writeData(val:=Value);
END_IF;
resetCommand();

PROPERTY archSrcValue : REAL
GET
END_GET
END_PROPERTY

PROPERTY archValue : REAL
GET
archValue:=value;
END_GET
END_PROPERTY

METHOD PRIVATE cmdSetValue
VAR_INPUT
	nValue:REAL;
END_VAR
setCmd(cmd_ChangeValue);
setValue(nValue:=nValue);
END_METHOD

{attribute 'symbol' := 'none'}
PROPERTY imit : BOOL
GET
imit:=_imit;
END_GET
SET
_imit:=imit;
END_SET
END_PROPERTY

METHOD PROTECTED processCmd;
VAR_INPUT
	cmd:UINT;
	sender:UINT;
	parametr:UINT;
END_VAR
CASE cmd OF
	cmd_ChangeValue:cmdSetValue(newValue);
	cmd_ChangeLimits:setLimits();
END_CASE
END_METHOD

METHOD PROTECTED readPersistent
VAR_INPUT
END_VAR
Ll:=FPU.StrToReal(readValue());
Hl:=FPU.StrToReal(readValue());
END_METHOD

METHOD PROTECTED setDefaultPersistent:BOOL
VAR_INPUT
END_VAR
LL:=dLL;
Hl:=dHL;
setDefaultPersistent:=TRUE;
END_METHOD

METHOD setLimits
VAR_INPUT
END_VAR
setCmd(nCmd:=cmd_ChangeLimits);
Ll:=newLl;
Hl:=newHl;

SaveToFile();
END_METHOD

METHOD PUBLIC setValue
VAR_INPUT
	nValue:REAL;
END_VAR
IF ((FPU.IsRealNaN(Ll))OR(nValue>=Ll)) AND ((FPU.IsRealNaN(Hl))OR(nValue<=Hl) ) THEN
	Value:=nValue;
END_IF
END_METHOD

METHOD PROTECTED writeData
VAR_INPUT
	val:REAL;
END_VAR
END_METHOD

METHOD PROTECTED writePersistent
VAR_INPUT
END_VAR
writeValue(value:=FPU.RealToStr(LL),comment:='LL');
writeValue(value:=FPU.RealToStr(Hl),comment:='HL');
END_METHOD

END_FUNCTION_BLOCK

// LowLevel_Algoritms/algoritms/AiProtectionDual
	{attribute 'symbol' := 'none'}
FUNCTION_BLOCK AiProtectionDual EXTENDS BaseProtection
VAR_INPUT
	ai1:REFERENCE TO AISource;
	ai2:REFERENCE TO AISource;
	controlLimit:statusAi;
	control_Normal:statusAi;
	{attribute 'symbol' := 'read'}
	delay:TimeParametr(table:=ADR(objectTable));	
END_VAR
VAR_OUTPUT
END_VAR
VAR
	timer:TON;
END_VAR

SUPER^();
IF __ISVALIDREF(ai1) AND __ISVALIDREF(ai2) THEN
	timer(IN:=(	((ai1.interval=controlLimit) AND (ai2.interval=controlLimit)) OR 
				((ai1.interval=controlLimit) AND (ai2.interval < control_Normal)) OR 
				((ai2.interval=controlLimit) AND (ai1.interval < control_Normal))),PT:=delay.Value);
	IF timer.Q THEN
		signaling:=TRUE; 
	ELSE
		signaling:=FALSE;
	END_IF
END_IF

METHOD PUBLIC reset
VAR_INPUT
END_VAR
SUPER^.reset();
timer(in:=FALSE);
signaling:=FALSE;
END_METHOD

END_FUNCTION_BLOCK

// lowLevel_ecl/algoritms/BaseProtection
	{attribute 'symbol' := 'none'}
FUNCTION_BLOCK BaseProtection EXTENDS BaseAlgoritm IMPLEMENTS IProtection
VAR_INPUT
END_VAR
VAR_OUTPUT
	
END_VAR
VAR
	_remont:BOOL;
	_signaling:BOOL;
	_check:BOOL;
	
	_signalingTp:TOF:=(PT:=T#1s);
END_VAR
VAR CONSTANT
	cmd_check:UINT:=3;
	cmd_setRemont:UINT:=4;
	cmd_resetRemont:UINT:=5;
END_VAR

SUPER^();

METHOD PUBLIC check
VAR_INPUT
END_VAR
setCmd(nCmd:=cmd_check);
_check:=TRUE;
resetCommand();
END_METHOD

METHOD PROTECTED processCmd;
VAR_INPUT
	cmd:UINT;
	sender:UINT;
	parametr:UINT;
END_VAR
SUPER^.processCmd(cmd,sender,parametr);
CASE cmd OF
	cmd_SetRemont:setRemont();
	cmd_ResetRemont:resetRemont();
END_CASE
END_METHOD

METHOD PROTECTED readPersistent
VAR_INPUT
END_VAR
SUPER^.readPersistent();
_remont:=STRING_TO_BOOL(readValue());
IF remont THEN
	reset();
END_IF
END_METHOD

PROPERTY PUBLIC remont : BOOL
GET
remont:=_remont;
END_GET
SET
PRIVATE
VAR
END_VAR
IF (NOT remont) AND (_signaling) THEN
	signaling:=FALSE;
	THIS^();
END_IF
IF ((NOT _signaling) OR (remont)) THEN
	_remont:=remont;
END_IF
END_SET
END_PROPERTY

METHOD reset
VAR_INPUT
END_VAR
VAR
	curObject:POINTER TO BaseObject;
	curPhase:IAlgoritmPhase;
END_VAR
signaling:=FALSE;
_check:=FALSE;
SUPER^.reset();
END_METHOD

METHOD PUBLIC resetRemont
VAR_INPUT
END_VAR
setCmd(nCmd:=cmd_resetRemont);
remont:=FALSE;
IF (NOT remont) THEN
	resetCommand();
ELSE
	errorCommand();
END_IF
END_METHOD

METHOD PUBLIC run
VAR_INPUT
END_VAR
IF (NOT remont) THEN
	SUPER^.run();
ELSE
	setCmd(nCmd:=cmdRun);
	errorCommand();	
END_IF
END_METHOD

METHOD PUBLIC setRemont
VAR_INPUT
END_VAR
setCmd(nCmd:=cmd_setRemont);
remont:=TRUE;
resetCommand();
END_METHOD

PROPERTY PUBLIC signaling : BOOL
GET
IF (NOT remont) AND (NOT _check) THEN
	signaling:=_signaling;
ELSE
	signaling:=FALSE;
END_IF
END_GET
SET
PROTECTED 
VAR
END_VAR
_signaling:=signaling;
IF NOT remont THEN
	_signalingTp(in:=_signaling);
ELSE
	_signalingTp(in:=FALSE);
END_IF
END_SET
END_PROPERTY

METHOD PUBLIC writeImStatus
VAR_INPUT
END_VAR
SUPER^.writeImStatus();
_signalingTp();
statusSet.setBit(3,_signalingTp.Q);
statusSet.setBit(5,_check);
statusSet.setBit(6,remont);
END_METHOD

METHOD PROTECTED writePersistent
VAR_INPUT
END_VAR
SUPER^.writePersistent();
writeValue(value:=BOOL_TO_STRING(_remont),comment:='Ремонт');
END_METHOD

END_FUNCTION_BLOCK

// lowLevel_ecl/algoritms/BaseAlgoritm
	{attribute 'symbol' := 'none'}
FUNCTION_BLOCK BaseAlgoritm EXTENDS BaseIm
IMPLEMENTS AlgoritmInterface
VAR_INPUT
	runOnStart:BOOL:=FALSE;
END_VAR
VAR_OUTPUT
END_VAR
VAR
	_runing:BOOL;
	_ended:BOOL;
	_CanRun: BOOL:=TRUE;
	_hasError:BOOL;
END_VAR
VAR CONSTANT
	cmdRun:WORD:=1;
	cmdReset:WORD:=2;
END_VAR

//Вызов Super^() сдесь не нужен

PROPERTY autoRun : bool
GET
autoRun:=runOnStart;
END_GET
END_PROPERTY

METHOD PUBLIC FINAL callBase
VAR_INPUT
END_VAR
VAR

END_VAR
SUPER^();
writeImStatus();
END_METHOD

PROPERTY CanRun : BOOL
GET
CanRun:=_CanRun;
END_GET
SET
_CanRun:=CanRun;
END_SET
END_PROPERTY

METHOD PROTECTED end
VAR_INPUT
END_VAR
_ended:=true;
END_METHOD

METHOD PUBLIC getTable :POINTER TO TableDescriptor
VAR_INPUT
END_VAR
getTable:=adr(objectTable);
END_METHOD

PROPERTY PUBLIC hasError : bool
GET
hasError:=_hasError;
END_GET
SET
PROTECTED 
VAR
END_VAR
_hasError:=hasError;
END_SET
END_PROPERTY

PROPERTY PUBLIC isEnded : bool
GET
isEnded:=_ended;
END_GET
END_PROPERTY

PROPERTY isRuning : BOOL
GET
isRuning:=_runing;
END_GET
END_PROPERTY

METHOD PROTECTED onInit
VAR_INPUT
END_VAR
VAR
	curObject:POINTER TO BaseObject;
	IcurAlg:AlgoritmInterface;
END_VAR
SUPER^.onInit();

curObject:=objectTable.head;
IF curObject<>0 THEN
	REPEAT
		IF (__QUERYINTERFACE(curObject^,IcurAlg)) THEN	
			IcurAlg.callBase();
			IcurAlg.reset();
			IF IcurAlg.autoRun THEN
				IcurAlg.run();
			END_IF
		END_IF;
		curObject:=curObject^.getNext();
	UNTIL curObject=0
	END_REPEAT;
END_IF;
END_METHOD

METHOD PROTECTED processCmd;
VAR_INPUT
	cmd:UINT;
	sender:UINT;
	parametr:UINT;
END_VAR
CASE cmd OF
	cmdRun:
		run();
	cmdReset:
		reset();
END_CASE
END_METHOD

METHOD PROTECTED processObjectTable
VAR_INPUT
END_VAR
VAR
		curObject:POINTER TO BaseObject;
		IcurAlg:AlgoritmInterface;
END_VAR
curObject:=objectTable.head;
IF curObject<>0 THEN
	REPEAT
		IF (__QUERYINTERFACE(curObject^,IcurAlg)) THEN
			IcurAlg.callBase();	
			IF IcurAlg.isRuning THEN	
				curObject^();
			END_IF;			
		ELSE
			callObject(curObject);			
		END_IF;
	
		curObject:=curObject^.getNext();
	UNTIL curObject=0
	END_REPEAT;
END_IF;
END_METHOD

METHOD reset
VAR_INPUT
END_VAR
VAR
	curObject:POINTER TO BaseObject;
	curPhase:IAlgoritmPhase;
END_VAR
setCmd(cmdReset);
end();
_runing:=FALSE;
_ended:=FALSE;
resetCommand();
END_METHOD

METHOD run
VAR_INPUT
END_VAR
VAR
	curObject:POINTER TO BaseObject;
	curPhase:IAlgoritmPhase;
END_VAR
setCmd(cmdRun);
IF (CanRun) THEN
	_runing:=TRUE;
	resetCommand();
ELSE
	errorCommand();
END_IF
END_METHOD

METHOD PUBLIC writeImStatus
VAR_INPUT
END_VAR
statusSet.setBit(0,isRuning);
statusSet.setBit(1,_ended);
statusSet.setBit(2,_canRun);
statusSet.setBit(4,hasError);
END_METHOD

END_FUNCTION_BLOCK

// lowLevel_ecl/algoritms/AlgoritmInterface
INTERFACE AlgoritmInterface EXTENDS __SYSTEM.IQueryInterface

PROPERTY autoRun : bool
GET
END_GET
END_PROPERTY

METHOD PUBLIC callBase
VAR_INPUT
END_VAR
END_METHOD

PROPERTY CanRun : bool
GET
END_GET
SET
END_SET
END_PROPERTY

PROPERTY isRuning : bool
GET
END_GET
END_PROPERTY

METHOD reset
VAR_INPUT
END_VAR
END_METHOD

METHOD run
VAR_INPUT
END_VAR
END_METHOD

END_INTERFACE

// lowLevel_ecl/algoritms/phases/IAlgoritmPhase
INTERFACE IAlgoritmPhase EXTENDS __SYSTEM.IQueryInterface

PROPERTY error : Bool
GET
END_GET
END_PROPERTY

METHOD getPhaseNum : UINT
VAR_INPUT
END_VAR
END_METHOD

METHOD reset : Bool
VAR_INPUT
END_VAR
END_METHOD

METHOD run
VAR_INPUT
END_VAR
END_METHOD

METHOD setBlockIm
VAR_INPUT
	algRuning:BOOL;
END_VAR
END_METHOD

PROPERTY start : Bool
GET
END_GET
END_PROPERTY

PROPERTY top : Bool
GET
END_GET
END_PROPERTY

END_INTERFACE

// lowLevel_ecl/algoritms/IProtection
INTERFACE IProtection

METHOD PUBLIC check
VAR_INPUT
END_VAR
END_METHOD

PROPERTY PUBLIC remont : BOOL
GET
END_GET
END_PROPERTY

PROPERTY PUBLIC signaling : BOOL
GET
END_GET
END_PROPERTY

END_INTERFACE

// lowLevel_ecl/Common/parameters/TimeParametr
	{attribute 'symbol' := 'none'}
FUNCTION_BLOCK TimeParametr EXTENDS BaseIm
VAR_INPUT
		{attribute 'symbol' := 'readwrite'}
	newValue:TIME;	
END_VAR
VAR_OUTPUT
		{attribute 'symbol' := 'read'}
	Value:TIME;
END_VAR
VAR
	
END_VAR
VAR CONSTANT
	cmd_ChangeValue:WORD:=1;
END_VAR


SUPER^();

resetCommand();

METHOD PROTECTED processCmd;
VAR_INPUT
	cmd:UINT;
	sender:UINT;
	parametr:UINT;
END_VAR
CASE cmd OF
	cmd_ChangeValue:setValue(newValue);
END_CASE
END_METHOD

METHOD PROTECTED readPersistent
VAR_INPUT
END_VAR
Value:=STRING_TO_TIME(readValue());
END_METHOD

METHOD PUBLIC setValue
VAR_INPUT
	nValue:TIME;
END_VAR
setCmd(cmd_ChangeValue);
Value:=nValue;

SaveToFile();
END_METHOD

METHOD PROTECTED writePersistent
VAR_INPUT
END_VAR
writeValue(value:=TIME_TO_STRING(Value),comment:='value');
END_METHOD

END_FUNCTION_BLOCK

// K1/std12k5/AlgoritmsManager
	{attribute 'symbol' := 'none'}
FUNCTION_BLOCK AlgoritmsManager EXTENDS BaseAlgoritmsManager
VAR_INPUT
END_VAR
VAR_OUTPUT
	{attribute 'symbol' := 'read'}
	mode:ModeGpa;
	reg_V:BOOL;
END_VAR
VAR
	AoTrig:F_TRIG;
END_VAR

SUPER^();

METHOD PROTECTED onStart
VAR_INPUT
END_VAR
algoritms.opcComands.CanRun:=TRUE;
algoritms.opcComands.run();
///*ТЕМПЕРАТУРЫ*///////
(*Температуры т.1 - т.10*) 
		protections.p_TOpornogoPodshipnikaEDT_1.run();
		protections.p_TOpornoYpornogoPodshipnikaEDT_2.run();
		protections.p_TOpornoYpornogoPodshipnikaKolesaRedEDT_3.run();
		protections.p_TOpornoYpornogoPodshipnikaKolesaRedHT_4.run();
		protections.p_TOpornogoPodshipnikaShesterniReduktoraT_5.run();
		protections.p_TOpornogoPodshipnikaReduktoraHT_6.run();
		protections.p_TOpornoYpornogoPodshipnikaNagnetateljaT_7.run();
																										
		protections.p_TOpornoYpornogoPodshipnikaSvobodnogoKoncaNT_8.run();
		protections.p_TYpornogoPodshipnikaRavKolodokHT_9.run();
		protections.p_TYpornogoPodshipnikaNerabKolodokHT_10.run();
		protections.p_TgazaNaVyhodeH.run();
		
	(*Давления*)
		
		protections.p_OsSdvigNagnetatelja_Plus.run();
		protections.p_OsSdvigNagnetatelja_Minus.run();
		
	
	(*Дискретные сигналы *)
		
		
		protections.p_AO_PRU.run();
		protections.p_AO_fromSHU.run();
					
		algoritms.Synch_Rejim_.CanRun:=TRUE;
		algoritms.Synch_Rejim_.run ();
		
im.mv.DisableOpcControl ();
im.kran1.DisableOpcControl ();
im.kran2.DisableOpcControl ();
im.kran3.DisableOpcControl ();
im.kran3b.DisableOpcControl ();
im.kran4.DisableOpcControl ();
im.kran5.DisableOpcControl ();
END_METHOD

METHOD PROTECTED onInit
VAR_INPUT
END_VAR
VAR
	curObject:POINTER TO BaseObject;
	IcurAlg:AlgoritmInterface;
END_VAR
SUPER^.onInit();
setMode(nMode:=ModeGpa.MODE_STOP);
END_METHOD

METHOD PUBLIC setMode
VAR_INPUT
	nMode:ModeGpa;
END_VAR
IF 	nMode<>mode THEN
	mode:=nMode;
	CASE 	mode OF
	mode_stop:	resetAndDisable(alg:=algoritms.Auto_Avom_);
		resetAndDisable(alg:=algoritms.autoNu_1);
		resetAndDisable(alg:=algoritms.autoNu_2);
		resetAndDisable(alg:=algoritms.autoPns);
		resetAndDisable(alg:=algoritms.AUto_Ten_);
		resetAndDisable(alg:=algoritms.PNS_ON_MV_);
		resetAndDisable(alg:=algoritms.no);
		resetAndDisable(alg:=algoritms.ao);
		resetAndDisable(alg:=algoritms.Pms);
		resetAndDisable(alg:=algoritms.dPmg);
		resetAndDisable(alg:=algoritms.F1_1);
		resetAndDisable(alg:=algoritms.F1_2);
		resetAndDisable(alg:=algoritms.F2_Ch);
		resetAndDisable(alg:=algoritms.F2_R);
		resetAndDisable(alg:=algoritms.F3);
		resetAndDisable(alg:=algoritms.F4);
		resetAndDisable(alg:=algoritms.Kr6_Move);
		resetAndDisable(alg:=algoritms.AutoPNS_Start);
		resetAndDisable(alg:=algoritms.R_AutoAVom);
		resetAndDisable(alg:=algoritms.S_AutoAVOM);
		resetAndDisable(alg:=algoritms.S_Vibr);
		resetAndDisable(alg:=algoritms.S_dPmg);
		resetAndDisable(alg:=algoritms.S_I);
		resetAndDisable(alg:=algoritms.S_K);
		resetAndDisable(alg:=algoritms.S_Pms);
		resetAndDisable(alg:=algoritms.S_V);
		resetAndDisable(alg:=algoritms.S_AP);
		resetAndDisable(alg:=algoritms.S_PP);
		resetAndDisable(alg:=algoritms.Test_IM);
		algoritms.Opres.CanRun:=TRUE;
		algoritms.ppu.CanRun:=TRUE;
		resetAndDisable(alg:=algoritms.R_AutoTEN);
		//algoritms.R_AutoTEN.CanRun:=TRUE;
		algoritms.S_AutoTEN.CanRun:=TRUE;
		algoritms.S_Test_IM.CanRun:=TRUE;
		resetAndDisable(alg:=algoritms.R_TestIM);
		algoritms.S_NO.CanRun:=TRUE;
		algoritms.S_AO.CanRun:=TRUE;
		algmanager.reg_V:=FALSE;
		algoritms.Start_Test_P.CanRun:=TRUE;
		resetAndDisable(alg:=algoritms.Test_P);
		algoritms.Test_P.DisableOpcControl();
		
		////////////*АЛГОРИТМЫ РАБОТАЮЩИЕ В РЕЖИМЕ АВТОМАТИЧЕСКИЙ Реакторный  ПУСК*/////////////////////////////////
MODE_PUSKAP_R:
	resetAndDisable(alg:=algoritms.Auto_Avom_);
	resetAndDisable(alg:=algoritms.autoNu_1);
	resetAndDisable(alg:=algoritms.autoNu_2);
	resetAndDisable(alg:=algoritms.autoPns);
	resetAndDisable(alg:=algoritms.AUto_Ten_);
	resetAndDisable(alg:=algoritms.PNS_ON_MV_);
	resetAndDisable(alg:=algoritms.no);
	resetAndDisable(alg:=algoritms.ao);
	resetAndDisable(alg:=algoritms.Opres);
	resetAndDisable(alg:=algoritms.Pms);
	resetAndDisable(alg:=algoritms.dPmg);
	algoritms.ppu.CanRun:=TRUE;
	algoritms.ppu.run();
	resetAndDisable(alg:=algoritms.F1_2);
	resetAndDisable(alg:=algoritms.F2_Ch);
	resetAndDisable(alg:=algoritms.F2_R);
	resetAndDisable(alg:=algoritms.F3);
	resetAndDisable(alg:=algoritms.F4);
	resetAndDisable(alg:=algoritms.Kr6_Move);
	resetAndDisable(alg:=algoritms.AutoPNS_Start);
	resetAndDisable(alg:=algoritms.R_AutoAVom);
	resetAndDisable(alg:=algoritms.R_AutoTEN);
	resetAndDisable(alg:=algoritms.R_TestIM);
	resetAndDisable(alg:=algoritms.S_AutoAVOM);
	resetAndDisable(alg:=algoritms.S_AutoTEN);
	resetAndDisable(alg:=algoritms.S_Test_IM);
	resetAndDisable(alg:=algoritms.S_Vibr);
	resetAndDisable(alg:=algoritms.S_dPmg);
	resetAndDisable(alg:=algoritms.S_I);
	resetAndDisable(alg:=algoritms.S_K);
	resetAndDisable(alg:=algoritms.S_Pms);
	resetAndDisable(alg:=algoritms.S_V);
	resetAndDisable(alg:=algoritms.S_PP);
	algoritms.S_AP.CanRun:=FALSE;
	algoritms.S_NO.CanRun:=TRUE;
	algoritms.S_AO.CanRun:=TRUE;
	resetAndDisable(alg:=algoritms.Test_IM);
	resetAndDisable(alg:=algoritms.Start_Test_P);
	resetAndDisable(alg:=algoritms.Test_P);
MODE_PUSKAP_Ch:
	resetAndDisable(alg:=algoritms.Auto_Avom_);
	resetAndDisable(alg:=algoritms.autoNu_1);
	resetAndDisable(alg:=algoritms.autoNu_2);
	resetAndDisable(alg:=algoritms.autoPns);
	resetAndDisable(alg:=algoritms.AUto_Ten_);
	resetAndDisable(alg:=algoritms.PNS_ON_MV_);
	resetAndDisable(alg:=algoritms.no);
	resetAndDisable(alg:=algoritms.ao);
	resetAndDisable(alg:=algoritms.Opres);
	resetAndDisable(alg:=algoritms.Pms);
	resetAndDisable(alg:=algoritms.dPmg);
	algoritms.ppu.CanRun:=TRUE;
	algoritms.ppu.run();
	resetAndDisable(alg:=algoritms.F1_2);
	resetAndDisable(alg:=algoritms.F2_Ch);
	resetAndDisable(alg:=algoritms.F2_R);
	resetAndDisable(alg:=algoritms.F3);
	resetAndDisable(alg:=algoritms.F4);
	resetAndDisable(alg:=algoritms.Kr6_Move);
	resetAndDisable(alg:=algoritms.AutoPNS_Start);
	resetAndDisable(alg:=algoritms.R_AutoAVom);
	resetAndDisable(alg:=algoritms.R_AutoTEN);
	resetAndDisable(alg:=algoritms.R_TestIM);
	resetAndDisable(alg:=algoritms.S_AutoAVOM);
	resetAndDisable(alg:=algoritms.S_AutoTEN);
	resetAndDisable(alg:=algoritms.S_Test_IM);
	resetAndDisable(alg:=algoritms.S_Vibr);
	resetAndDisable(alg:=algoritms.S_dPmg);
	resetAndDisable(alg:=algoritms.S_I);
	resetAndDisable(alg:=algoritms.S_K);
	resetAndDisable(alg:=algoritms.S_Pms);
	resetAndDisable(alg:=algoritms.S_V);
	resetAndDisable(alg:=algoritms.S_PP);
	algoritms.S_AP.CanRun:=FALSE;
	algoritms.S_NO.CanRun:=TRUE;
	algoritms.S_AO.CanRun:=TRUE;
	resetAndDisable(alg:=algoritms.Test_IM);
	resetAndDisable(alg:=algoritms.Start_Test_P);
	resetAndDisable(alg:=algoritms.Test_P);
MODE_PUSKPP_R:
	resetAndDisable(alg:=algoritms.Auto_Avom_);
	resetAndDisable(alg:=algoritms.autoNu_1);
	resetAndDisable(alg:=algoritms.autoNu_2);
	resetAndDisable(alg:=algoritms.autoPns);
	resetAndDisable(alg:=algoritms.AUto_Ten_);
	resetAndDisable(alg:=algoritms.PNS_ON_MV_);
	resetAndDisable(alg:=algoritms.no);
	resetAndDisable(alg:=algoritms.ao);
	resetAndDisable(alg:=algoritms.Opres);
	resetAndDisable(alg:=algoritms.Pms);
	resetAndDisable(alg:=algoritms.dPmg);
	algoritms.ppu.CanRun:=TRUE;
	algoritms.ppu.run();
	resetAndDisable(alg:=algoritms.F1_2);
	resetAndDisable(alg:=algoritms.F2_Ch);
	resetAndDisable(alg:=algoritms.F2_R);
	resetAndDisable(alg:=algoritms.F3);
	resetAndDisable(alg:=algoritms.F4);
	resetAndDisable(alg:=algoritms.Kr6_Move);
	resetAndDisable(alg:=algoritms.AutoPNS_Start);
	resetAndDisable(alg:=algoritms.R_AutoAVom);
	resetAndDisable(alg:=algoritms.R_AutoTEN);
	resetAndDisable(alg:=algoritms.R_TestIM);
	resetAndDisable(alg:=algoritms.S_AutoAVOM);
	resetAndDisable(alg:=algoritms.S_AutoTEN);
	resetAndDisable(alg:=algoritms.S_Test_IM);
	resetAndDisable(alg:=algoritms.S_Vibr);
	resetAndDisable(alg:=algoritms.S_dPmg);
	resetAndDisable(alg:=algoritms.S_I);
	resetAndDisable(alg:=algoritms.S_K);
	resetAndDisable(alg:=algoritms.S_Pms);
	resetAndDisable(alg:=algoritms.S_V);
	resetAndDisable(alg:=algoritms.S_AP);
	algoritms.S_PP.CanRun:=FALSE;
	algoritms.S_NO.CanRun:=TRUE;
	algoritms.S_AO.CanRun:=TRUE;
	resetAndDisable(alg:=algoritms.Test_IM);
	resetAndDisable(alg:=algoritms.Start_Test_P);
	resetAndDisable(alg:=algoritms.Test_P);
MODE_PUSKPP_Ch:
	resetAndDisable(alg:=algoritms.Auto_Avom_);
	resetAndDisable(alg:=algoritms.autoNu_1);
	resetAndDisable(alg:=algoritms.autoNu_2);
	resetAndDisable(alg:=algoritms.autoPns);
	resetAndDisable(alg:=algoritms.AUto_Ten_);
	resetAndDisable(alg:=algoritms.PNS_ON_MV_);
	resetAndDisable(alg:=algoritms.no);
	resetAndDisable(alg:=algoritms.ao);
	resetAndDisable(alg:=algoritms.Opres);
	resetAndDisable(alg:=algoritms.Pms);
	resetAndDisable(alg:=algoritms.dPmg);
	algoritms.ppu.CanRun:=TRUE;
	algoritms.ppu.run();
	resetAndDisable(alg:=algoritms.F1_2);
	resetAndDisable(alg:=algoritms.F2_Ch);
	resetAndDisable(alg:=algoritms.F2_R);
	resetAndDisable(alg:=algoritms.F3);
	resetAndDisable(alg:=algoritms.F4);
	resetAndDisable(alg:=algoritms.Kr6_Move);
	resetAndDisable(alg:=algoritms.AutoPNS_Start);
	resetAndDisable(alg:=algoritms.R_AutoAVom);
	resetAndDisable(alg:=algoritms.R_AutoTEN);
	resetAndDisable(alg:=algoritms.R_TestIM);
	resetAndDisable(alg:=algoritms.S_AutoAVOM);
	resetAndDisable(alg:=algoritms.S_AutoTEN);
	resetAndDisable(alg:=algoritms.S_Test_IM);
	resetAndDisable(alg:=algoritms.S_Vibr);
	resetAndDisable(alg:=algoritms.S_dPmg);
	resetAndDisable(alg:=algoritms.S_I);
	resetAndDisable(alg:=algoritms.S_K);
	resetAndDisable(alg:=algoritms.S_Pms);
	resetAndDisable(alg:=algoritms.S_V);
	resetAndDisable(alg:=algoritms.S_AP);
	algoritms.S_PP.CanRun:=FALSE;
	algoritms.S_NO.CanRun:=TRUE;
	algoritms.S_AO.CanRun:=TRUE;
	resetAndDisable(alg:=algoritms.Test_IM);
	resetAndDisable(alg:=algoritms.Start_Test_P);
	resetAndDisable(alg:=algoritms.Test_P);
MODE_WORK_M:
	resetAndDisable(alg:=algoritms.autoNu_1);
	resetAndDisable(alg:=algoritms.AUto_Ten_);
	resetAndDisable(alg:=algoritms.PNS_ON_MV_);
	resetAndDisable(alg:=algoritms.no);
	resetAndDisable(alg:=algoritms.ao);
	resetAndDisable(alg:=algoritms.Opres);
	resetAndDisable(alg:=algoritms.Pms);
	resetAndDisable(alg:=algoritms.dPmg);
	algoritms.ppu.CanRun:=TRUE;
	algoritms.ppu.run();
	resetAndDisable(alg:=algoritms.F1_1);
	resetAndDisable(alg:=algoritms.F1_2);
	resetAndDisable(alg:=algoritms.F2_Ch);
	resetAndDisable(alg:=algoritms.F2_R);
	resetAndDisable(alg:=algoritms.F3);
	resetAndDisable(alg:=algoritms.F4);
	resetAndDisable(alg:=algoritms.R_AutoTEN);
	resetAndDisable(alg:=algoritms.R_TestIM);
	resetAndDisable(alg:=algoritms.S_AutoTEN);
	resetAndDisable(alg:=algoritms.S_Test_IM);
	resetAndDisable(alg:=algoritms.S_dPmg);
	resetAndDisable(alg:=algoritms.S_I);
	resetAndDisable(alg:=algoritms.S_K);
	resetAndDisable(alg:=algoritms.S_Pms);
	resetAndDisable(alg:=algoritms.S_V);
	resetAndDisable(alg:=algoritms.S_AP);
	resetAndDisable(alg:=algoritms.S_PP);
	algoritms.S_NO.CanRun:=TRUE;
	algoritms.S_AO.CanRun:=TRUE;
	resetAndDisable(alg:=algoritms.Test_IM);
	resetAndDisable(alg:=algoritms.Start_Test_P);
	resetAndDisable(alg:=algoritms.Test_P);
MODE_WORK_K:
	resetAndDisable(alg:=algoritms.autoNu_1);
	resetAndDisable(alg:=algoritms.AUto_Ten_);
	resetAndDisable(alg:=algoritms.PNS_ON_MV_);
	resetAndDisable(alg:=algoritms.no);
	resetAndDisable(alg:=algoritms.ao);
	resetAndDisable(alg:=algoritms.Opres);
	resetAndDisable(alg:=algoritms.Pms);
	resetAndDisable(alg:=algoritms.dPmg);
	algoritms.ppu.CanRun:=TRUE;
	algoritms.ppu.run();
	resetAndDisable(alg:=algoritms.F1_1);
	resetAndDisable(alg:=algoritms.F1_2);
	resetAndDisable(alg:=algoritms.F2_Ch);
	resetAndDisable(alg:=algoritms.F2_R);
	resetAndDisable(alg:=algoritms.F3);
	resetAndDisable(alg:=algoritms.F4);
	resetAndDisable(alg:=algoritms.R_AutoTEN);
	resetAndDisable(alg:=algoritms.R_TestIM);
	resetAndDisable(alg:=algoritms.S_AutoTEN);
	resetAndDisable(alg:=algoritms.S_Test_IM);
	resetAndDisable(alg:=algoritms.S_dPmg);
	resetAndDisable(alg:=algoritms.S_I);
	resetAndDisable(alg:=algoritms.S_K);
	resetAndDisable(alg:=algoritms.S_Pms);
	resetAndDisable(alg:=algoritms.S_V);
	resetAndDisable(alg:=algoritms.S_AP);
	resetAndDisable(alg:=algoritms.S_PP);
	algoritms.S_NO.CanRun:=TRUE;
	algoritms.S_AO.CanRun:=TRUE;
	resetAndDisable(alg:=algoritms.Test_IM);
	resetAndDisable(alg:=algoritms.Start_Test_P);
	resetAndDisable(alg:=algoritms.Test_P);
MODE_NO:
		resetAndDisable(alg:=algoritms.AUto_Ten_);
		resetAndDisable(alg:=algoritms.PNS_ON_MV_);
		resetAndDisable(alg:=algoritms.ao);
		resetAndDisable(alg:=algoritms.Opres);
		resetAndDisable(alg:=algoritms.Pms);
		resetAndDisable(alg:=algoritms.dPmg);
		resetAndDisable(alg:=algoritms.ppu);
		resetAndDisable(alg:=algoritms.F1_1);
		resetAndDisable(alg:=algoritms.F1_2);
		resetAndDisable(alg:=algoritms.F2_Ch);
		resetAndDisable(alg:=algoritms.F2_R);
		resetAndDisable(alg:=algoritms.F3);
		resetAndDisable(alg:=algoritms.F4);
		resetAndDisable(alg:=algoritms.Kr6_Move);
		resetAndDisable(alg:=algoritms.AutoPNS_Start);
		//resetAndDisable(alg:=algoritms.R_AutoAVom);
		resetAndDisable(alg:=algoritms.R_AutoTEN);
		resetAndDisable(alg:=algoritms.R_TestIM);
		//resetAndDisable(alg:=algoritms.S_AutoAVOM);
		resetAndDisable(alg:=algoritms.S_AutoTEN);
		resetAndDisable(alg:=algoritms.S_Test_IM);
		resetAndDisable(alg:=algoritms.S_dPmg);
		resetAndDisable(alg:=algoritms.S_I);
		resetAndDisable(alg:=algoritms.S_K);
		resetAndDisable(alg:=algoritms.S_Pms);
		resetAndDisable(alg:=algoritms.S_V);
		resetAndDisable(alg:=algoritms.S_AP);
		resetAndDisable(alg:=algoritms.S_PP);
		resetAndDisable(alg:=algoritms.S_NO);
		algoritms.S_AO.CanRun:=TRUE;
		resetAndDisable(alg:=algoritms.Test_IM);
		resetAndDisable(alg:=algoritms.Start_Test_P);
	resetAndDisable(alg:=algoritms.Test_P);
MODE_AO:
		resetAndDisable(alg:=algoritms.AUto_Ten_);
		resetAndDisable(alg:=algoritms.PNS_ON_MV_);
		resetAndDisable(alg:=algoritms.no);
		resetAndDisable(alg:=algoritms.Opres);
		resetAndDisable(alg:=algoritms.Pms);
		resetAndDisable(alg:=algoritms.dPmg);
		resetAndDisable(alg:=algoritms.ppu);
		resetAndDisable(alg:=algoritms.F1_1);
		resetAndDisable(alg:=algoritms.F1_2);
		resetAndDisable(alg:=algoritms.F2_Ch);
		resetAndDisable(alg:=algoritms.F2_R);
		resetAndDisable(alg:=algoritms.F3);
		resetAndDisable(alg:=algoritms.F4);
		resetAndDisable(alg:=algoritms.Kr6_Move);
		resetAndDisable(alg:=algoritms.AutoPNS_Start);
		//resetAndDisable(alg:=algoritms.R_AutoAVom);
		resetAndDisable(alg:=algoritms.R_AutoTEN);
		resetAndDisable(alg:=algoritms.R_TestIM);
		//resetAndDisable(alg:=algoritms.S_AutoAVOM);
		resetAndDisable(alg:=algoritms.S_AutoTEN);
		resetAndDisable(alg:=algoritms.S_Test_IM);
		resetAndDisable(alg:=algoritms.S_dPmg);
		resetAndDisable(alg:=algoritms.S_I);
		resetAndDisable(alg:=algoritms.S_K);
		resetAndDisable(alg:=algoritms.S_Pms);
		resetAndDisable(alg:=algoritms.S_V);
		resetAndDisable(alg:=algoritms.S_AP);
		resetAndDisable(alg:=algoritms.S_PP);
		resetAndDisable(alg:=algoritms.S_NO);
		resetAndDisable(alg:=algoritms.S_AO);
		resetAndDisable(alg:=algoritms.Test_IM);
		resetAndDisable(alg:=algoritms.Start_Test_P);
	resetAndDisable(alg:=algoritms.Test_P);
MODE_EO:		
		resetAndDisable(alg:=algoritms.Auto_Avom_);
		resetAndDisable(alg:=algoritms.autoNu_1);
		resetAndDisable(alg:=algoritms.autoNu_2);
		resetAndDisable(alg:=algoritms.autoPns);
		resetAndDisable(alg:=algoritms.AUto_Ten_);
		resetAndDisable(alg:=algoritms.PNS_ON_MV_);
		resetAndDisable(alg:=algoritms.no);
		resetAndDisable(alg:=algoritms.ao);
		resetAndDisable(alg:=algoritms.Opres);
		resetAndDisable(alg:=algoritms.Pms);
		resetAndDisable(alg:=algoritms.dPmg);
		resetAndDisable(alg:=algoritms.ppu);
		resetAndDisable(alg:=algoritms.F1_1);
		resetAndDisable(alg:=algoritms.F1_2);
		resetAndDisable(alg:=algoritms.F2_Ch);
		resetAndDisable(alg:=algoritms.F2_R);
		resetAndDisable(alg:=algoritms.F3);
		resetAndDisable(alg:=algoritms.F4);
		resetAndDisable(alg:=algoritms.Kr6_Move);
		resetAndDisable(alg:=algoritms.AutoPNS_Start);
		resetAndDisable(alg:=algoritms.R_AutoAVom);
		resetAndDisable(alg:=algoritms.R_AutoTEN);
		resetAndDisable(alg:=algoritms.R_TestIM);
		resetAndDisable(alg:=algoritms.S_AutoAVOM);
		resetAndDisable(alg:=algoritms.S_AutoTEN);
		resetAndDisable(alg:=algoritms.S_Test_IM);
		resetAndDisable(alg:=algoritms.S_Vibr);
		resetAndDisable(alg:=algoritms.S_dPmg);
		resetAndDisable(alg:=algoritms.S_I);
		resetAndDisable(alg:=algoritms.S_K);
		resetAndDisable(alg:=algoritms.S_Pms);
		resetAndDisable(alg:=algoritms.S_V);
		resetAndDisable(alg:=algoritms.S_AP);
		resetAndDisable(alg:=algoritms.S_PP);
		resetAndDisable(alg:=algoritms.S_NO);
		resetAndDisable(alg:=algoritms.S_AO);
		resetAndDisable(alg:=algoritms.Test_IM);
		Reset_ALL_P ();
		resetAndDisable(alg:=algoritms.Start_Test_P);
	resetAndDisable(alg:=algoritms.Test_P);

MODE_NOTDEFINED:		
		resetAndDisable(alg:=algoritms.Auto_Avom_);
		resetAndDisable(alg:=algoritms.autoNu_1);
		resetAndDisable(alg:=algoritms.autoNu_2);
		resetAndDisable(alg:=algoritms.autoPns);
		resetAndDisable(alg:=algoritms.AUto_Ten_);
		resetAndDisable(alg:=algoritms.PNS_ON_MV_);
		resetAndDisable(alg:=algoritms.no);
		resetAndDisable(alg:=algoritms.ao);
		resetAndDisable(alg:=algoritms.Opres);
		resetAndDisable(alg:=algoritms.Pms);
		resetAndDisable(alg:=algoritms.dPmg);
		resetAndDisable(alg:=algoritms.ppu);
		resetAndDisable(alg:=algoritms.F1_1);
		resetAndDisable(alg:=algoritms.F1_2);
		resetAndDisable(alg:=algoritms.F2_Ch);
		resetAndDisable(alg:=algoritms.F2_R);
		resetAndDisable(alg:=algoritms.F3);
		resetAndDisable(alg:=algoritms.F4);
		resetAndDisable(alg:=algoritms.Kr6_Move);
		resetAndDisable(alg:=algoritms.AutoPNS_Start);
		resetAndDisable(alg:=algoritms.R_AutoAVom);
		resetAndDisable(alg:=algoritms.R_AutoTEN);
		resetAndDisable(alg:=algoritms.R_TestIM);
		resetAndDisable(alg:=algoritms.S_AutoAVOM);
		resetAndDisable(alg:=algoritms.S_AutoTEN);
		resetAndDisable(alg:=algoritms.S_Test_IM);
		resetAndDisable(alg:=algoritms.S_Vibr);
		resetAndDisable(alg:=algoritms.S_dPmg);
		resetAndDisable(alg:=algoritms.S_I);
		resetAndDisable(alg:=algoritms.S_K);
		resetAndDisable(alg:=algoritms.S_Pms);
		resetAndDisable(alg:=algoritms.S_V);
		resetAndDisable(alg:=algoritms.S_AP);
		resetAndDisable(alg:=algoritms.S_PP);
		resetAndDisable(alg:=algoritms.S_NO);
		resetAndDisable(alg:=algoritms.S_AO);
		resetAndDisable(alg:=algoritms.Test_IM);
		resetAndDisable(alg:=algoritms.Start_Test_P);
	resetAndDisable(alg:=algoritms.Test_P);
MODE_TESTIM:
		resetAndDisable(alg:=algoritms.Auto_Avom_);
		resetAndDisable(alg:=algoritms.autoNu_1);
		resetAndDisable(alg:=algoritms.autoNu_2);
		resetAndDisable(alg:=algoritms.autoPns);
		resetAndDisable(alg:=algoritms.AUto_Ten_);
		resetAndDisable(alg:=algoritms.PNS_ON_MV_);
		resetAndDisable(alg:=algoritms.Opres);
		resetAndDisable(alg:=algoritms.Pms);
		resetAndDisable(alg:=algoritms.dPmg);
		resetAndDisable(alg:=algoritms.no);
		resetAndDisable(alg:=algoritms.ao);
		resetAndDisable(alg:=algoritms.ppu);
		resetAndDisable(alg:=algoritms.F1_1);
		resetAndDisable(alg:=algoritms.F1_2);
		resetAndDisable(alg:=algoritms.F2_Ch);
		resetAndDisable(alg:=algoritms.F2_R);
		resetAndDisable(alg:=algoritms.F3);
		resetAndDisable(alg:=algoritms.F4);
		resetAndDisable(alg:=algoritms.Kr6_Move);
		resetAndDisable(alg:=algoritms.AutoPNS_Start);
		resetAndDisable(alg:=algoritms.R_AutoAVom);
		resetAndDisable(alg:=algoritms.R_AutoTEN);
		algoritms.R_TestIM.CanRun:=TRUE;
		resetAndDisable(alg:=algoritms.S_AutoAVOM);
		resetAndDisable(alg:=algoritms.S_AutoTEN);
		resetAndDisable(alg:=algoritms.S_Test_IM);
		resetAndDisable(alg:=algoritms.S_Vibr);
		resetAndDisable(alg:=algoritms.S_dPmg);
		resetAndDisable(alg:=algoritms.S_I);
		resetAndDisable(alg:=algoritms.S_K);
		resetAndDisable(alg:=algoritms.S_Pms);
		resetAndDisable(alg:=algoritms.S_V);
		resetAndDisable(alg:=algoritms.S_AP);
		resetAndDisable(alg:=algoritms.S_PP);
		algoritms.S_NO.CanRun:=TRUE;
		algoritms.S_AO.CanRun:=TRUE;
		resetAndDisable(alg:=algoritms.Start_Test_P);
		resetAndDisable(alg:=algoritms.Test_P);
MODE_PUSKV_R:
	resetAndDisable(alg:=algoritms.Auto_Avom_);
	resetAndDisable(alg:=algoritms.autoNu_1);
	resetAndDisable(alg:=algoritms.autoNu_2);
	resetAndDisable(alg:=algoritms.autoPns);
	resetAndDisable(alg:=algoritms.AUto_Ten_);
	resetAndDisable(alg:=algoritms.PNS_ON_MV_);
	resetAndDisable(alg:=algoritms.no);
		resetAndDisable(alg:=algoritms.ao);
	resetAndDisable(alg:=algoritms.Opres);
	resetAndDisable(alg:=algoritms.Pms);
	resetAndDisable(alg:=algoritms.dPmg);
	algoritms.ppu.CanRun:=TRUE;
	algoritms.ppu.run();
	resetAndDisable(alg:=algoritms.F1_2);
	resetAndDisable(alg:=algoritms.F2_Ch);
	resetAndDisable(alg:=algoritms.F2_R);
	resetAndDisable(alg:=algoritms.F3);
	resetAndDisable(alg:=algoritms.F4);
	resetAndDisable(alg:=algoritms.Kr6_Move);
	resetAndDisable(alg:=algoritms.AutoPNS_Start);
	resetAndDisable(alg:=algoritms.R_AutoAVom);
	resetAndDisable(alg:=algoritms.R_AutoTEN);
	resetAndDisable(alg:=algoritms.R_TestIM);
	resetAndDisable(alg:=algoritms.S_AutoAVOM);
	resetAndDisable(alg:=algoritms.S_AutoTEN);
	resetAndDisable(alg:=algoritms.S_Test_IM);
	resetAndDisable(alg:=algoritms.S_Vibr);
	resetAndDisable(alg:=algoritms.S_dPmg);
	resetAndDisable(alg:=algoritms.S_I);
	resetAndDisable(alg:=algoritms.S_K);
	resetAndDisable(alg:=algoritms.S_Pms);
	algoritms.S_V.CanRun:=FALSE;
	resetAndDisable(alg:=algoritms.S_PP);
	resetAndDisable(alg:=algoritms.S_AP);
	algoritms.S_NO.CanRun:=TRUE;
	algoritms.S_AO.CanRun:=TRUE;
	resetAndDisable(alg:=algoritms.Test_IM);
	reg_V:=TRUE;
	resetAndDisable(alg:=algoritms.Start_Test_P);
		resetAndDisable(alg:=algoritms.Test_P);
MODE_PUSKV_Ch:
	resetAndDisable(alg:=algoritms.Auto_Avom_);
	resetAndDisable(alg:=algoritms.autoNu_1);
	resetAndDisable(alg:=algoritms.autoNu_2);
	resetAndDisable(alg:=algoritms.autoPns);
	resetAndDisable(alg:=algoritms.AUto_Ten_);
	resetAndDisable(alg:=algoritms.PNS_ON_MV_);
	resetAndDisable(alg:=algoritms.no);
		resetAndDisable(alg:=algoritms.ao);
	resetAndDisable(alg:=algoritms.Opres);
	resetAndDisable(alg:=algoritms.Pms);
	resetAndDisable(alg:=algoritms.dPmg);
	algoritms.ppu.CanRun:=TRUE;
	algoritms.ppu.run();
	resetAndDisable(alg:=algoritms.F1_2);
	resetAndDisable(alg:=algoritms.F2_Ch);
	resetAndDisable(alg:=algoritms.F2_R);
	resetAndDisable(alg:=algoritms.F3);
	resetAndDisable(alg:=algoritms.F4);
	resetAndDisable(alg:=algoritms.Kr6_Move);
	resetAndDisable(alg:=algoritms.AutoPNS_Start);
	resetAndDisable(alg:=algoritms.R_AutoAVom);
	resetAndDisable(alg:=algoritms.R_AutoTEN);
	resetAndDisable(alg:=algoritms.R_TestIM);
	resetAndDisable(alg:=algoritms.S_AutoAVOM);
	resetAndDisable(alg:=algoritms.S_AutoTEN);
	resetAndDisable(alg:=algoritms.S_Test_IM);
	resetAndDisable(alg:=algoritms.S_Vibr);
	resetAndDisable(alg:=algoritms.S_dPmg);
	resetAndDisable(alg:=algoritms.S_I);
	resetAndDisable(alg:=algoritms.S_K);
	resetAndDisable(alg:=algoritms.S_Pms);
	algoritms.S_V.CanRun:=FALSE;
	resetAndDisable(alg:=algoritms.S_PP);
	resetAndDisable(alg:=algoritms.S_AP);
	algoritms.S_NO.CanRun:=TRUE;
	algoritms.S_AO.CanRun:=TRUE;
	resetAndDisable(alg:=algoritms.Test_IM);
	reg_V:=TRUE;
	resetAndDisable(alg:=algoritms.Start_Test_P);
		resetAndDisable(alg:=algoritms.Test_P);
MODE_PUSKK:
	resetAndDisable(alg:=algoritms.Auto_Avom_);
	resetAndDisable(alg:=algoritms.autoNu_1);
	resetAndDisable(alg:=algoritms.autoNu_2);
	resetAndDisable(alg:=algoritms.autoPns);
	resetAndDisable(alg:=algoritms.AUto_Ten_);
	resetAndDisable(alg:=algoritms.PNS_ON_MV_);
	resetAndDisable(alg:=algoritms.no);
		resetAndDisable(alg:=algoritms.ao);
	resetAndDisable(alg:=algoritms.Opres);
	resetAndDisable(alg:=algoritms.Pms);
	resetAndDisable(alg:=algoritms.dPmg);
	algoritms.ppu.CanRun:=TRUE;
	algoritms.ppu.run();
	resetAndDisable(alg:=algoritms.F1_2);
	resetAndDisable(alg:=algoritms.F2_Ch);
	resetAndDisable(alg:=algoritms.F2_R);
	resetAndDisable(alg:=algoritms.F3);
	resetAndDisable(alg:=algoritms.F4);
	resetAndDisable(alg:=algoritms.Kr6_Move);
	resetAndDisable(alg:=algoritms.AutoPNS_Start);
	resetAndDisable(alg:=algoritms.R_AutoAVom);
	resetAndDisable(alg:=algoritms.R_AutoTEN);
	resetAndDisable(alg:=algoritms.R_TestIM);
	resetAndDisable(alg:=algoritms.S_AutoAVOM);
	resetAndDisable(alg:=algoritms.S_AutoTEN);
	resetAndDisable(alg:=algoritms.S_Test_IM);
	resetAndDisable(alg:=algoritms.S_Vibr);
	resetAndDisable(alg:=algoritms.S_dPmg);
	resetAndDisable(alg:=algoritms.S_I);
	algoritms.S_K.CanRun:=FALSE;
	resetAndDisable(alg:=algoritms.S_Pms);
	resetAndDisable(alg:=algoritms.S_V);
	resetAndDisable(alg:=algoritms.S_PP);
	resetAndDisable(alg:=algoritms.S_AP);
	algoritms.S_NO.CanRun:=TRUE;
	algoritms.S_AO.CanRun:=TRUE;
	resetAndDisable(alg:=algoritms.Test_IM);
	resetAndDisable(alg:=algoritms.Start_Test_P);
		resetAndDisable(alg:=algoritms.Test_P);
MODE_PROVPMS:
	resetAndDisable(alg:=algoritms.Auto_Avom_);
	resetAndDisable(alg:=algoritms.autoNu_1);
	resetAndDisable(alg:=algoritms.autoNu_2);
	resetAndDisable(alg:=algoritms.autoPns);
	resetAndDisable(alg:=algoritms.AUto_Ten_);
	resetAndDisable(alg:=algoritms.PNS_ON_MV_);
	resetAndDisable(alg:=algoritms.no);
		resetAndDisable(alg:=algoritms.ao);
	resetAndDisable(alg:=algoritms.Opres);
	resetAndDisable(alg:=algoritms.Pms);
	resetAndDisable(alg:=algoritms.dPmg);
	resetAndDisable(alg:=algoritms.ppu);
	resetAndDisable(alg:=algoritms.F1_2);
	resetAndDisable(alg:=algoritms.F2_Ch);
	resetAndDisable(alg:=algoritms.F2_R);
	resetAndDisable(alg:=algoritms.F3);
	resetAndDisable(alg:=algoritms.F4);
	resetAndDisable(alg:=algoritms.Kr6_Move);
	resetAndDisable(alg:=algoritms.AutoPNS_Start);
	resetAndDisable(alg:=algoritms.R_AutoAVom);
	resetAndDisable(alg:=algoritms.R_AutoTEN);
	resetAndDisable(alg:=algoritms.R_TestIM);
	resetAndDisable(alg:=algoritms.S_AutoAVOM);
	resetAndDisable(alg:=algoritms.S_AutoTEN);
	resetAndDisable(alg:=algoritms.S_Test_IM);
	resetAndDisable(alg:=algoritms.S_Vibr);
	resetAndDisable(alg:=algoritms.S_dPmg);
	resetAndDisable(alg:=algoritms.S_I);
	resetAndDisable(alg:=algoritms.S_K);
	algoritms.S_Pms.CanRun:=FALSE;
	resetAndDisable(alg:=algoritms.S_V);
	resetAndDisable(alg:=algoritms.S_PP);
	resetAndDisable(alg:=algoritms.S_AP);
	algoritms.S_NO.CanRun:=TRUE;
	algoritms.S_AO.CanRun:=TRUE;
	resetAndDisable(alg:=algoritms.Test_IM);
	resetAndDisable(alg:=algoritms.Start_Test_P);
		resetAndDisable(alg:=algoritms.Test_P);
MODE_PROBDPMG:
	resetAndDisable(alg:=algoritms.Auto_Avom_);
	resetAndDisable(alg:=algoritms.autoNu_1);
	resetAndDisable(alg:=algoritms.autoNu_2);
	resetAndDisable(alg:=algoritms.autoPns);
	resetAndDisable(alg:=algoritms.AUto_Ten_);
	resetAndDisable(alg:=algoritms.PNS_ON_MV_);
	resetAndDisable(alg:=algoritms.no);
		resetAndDisable(alg:=algoritms.ao);
	resetAndDisable(alg:=algoritms.Opres);
	resetAndDisable(alg:=algoritms.Pms);
	resetAndDisable(alg:=algoritms.dPmg);
	resetAndDisable(alg:=algoritms.ppu);
	resetAndDisable(alg:=algoritms.F1_2);
	resetAndDisable(alg:=algoritms.F2_Ch);
	resetAndDisable(alg:=algoritms.F2_R);
	resetAndDisable(alg:=algoritms.F3);
	resetAndDisable(alg:=algoritms.F4);
	resetAndDisable(alg:=algoritms.Kr6_Move);
	resetAndDisable(alg:=algoritms.AutoPNS_Start);
	resetAndDisable(alg:=algoritms.R_AutoAVom);
	resetAndDisable(alg:=algoritms.R_AutoTEN);
	resetAndDisable(alg:=algoritms.R_TestIM);
	resetAndDisable(alg:=algoritms.S_AutoAVOM);
	resetAndDisable(alg:=algoritms.S_AutoTEN);
	resetAndDisable(alg:=algoritms.S_Test_IM);
	resetAndDisable(alg:=algoritms.S_Vibr);
	resetAndDisable(alg:=algoritms.S_Pms);
	resetAndDisable(alg:=algoritms.S_I);
	resetAndDisable(alg:=algoritms.S_K);
	algoritms.S_dPmg.CanRun:=FALSE;
	resetAndDisable(alg:=algoritms.S_V);
	resetAndDisable(alg:=algoritms.S_PP);
	resetAndDisable(alg:=algoritms.S_AP);
	algoritms.S_NO.CanRun:=TRUE;
	algoritms.S_AO.CanRun:=TRUE;
	resetAndDisable(alg:=algoritms.Test_IM);
resetAndDisable(alg:=algoritms.Start_Test_P);
		resetAndDisable(alg:=algoritms.Test_P);
MODE_I:
	resetAndDisable(alg:=algoritms.Auto_Avom_);
	resetAndDisable(alg:=algoritms.autoNu_1);
	resetAndDisable(alg:=algoritms.autoNu_2);
	resetAndDisable(alg:=algoritms.autoPns);
	resetAndDisable(alg:=algoritms.AUto_Ten_);
	resetAndDisable(alg:=algoritms.PNS_ON_MV_);
	resetAndDisable(alg:=algoritms.no);
		resetAndDisable(alg:=algoritms.ao);
	resetAndDisable(alg:=algoritms.Opres);
	resetAndDisable(alg:=algoritms.Pms);
	resetAndDisable(alg:=algoritms.dPmg);
	algoritms.ppu.CanRun:=TRUE;
	algoritms.ppu.run();
	resetAndDisable(alg:=algoritms.F1_2);
	resetAndDisable(alg:=algoritms.F2_Ch);
	resetAndDisable(alg:=algoritms.F2_R);
	resetAndDisable(alg:=algoritms.F3);
	resetAndDisable(alg:=algoritms.F4);
	resetAndDisable(alg:=algoritms.Kr6_Move);
	resetAndDisable(alg:=algoritms.AutoPNS_Start);
	resetAndDisable(alg:=algoritms.R_AutoAVom);
	resetAndDisable(alg:=algoritms.R_AutoTEN);
	resetAndDisable(alg:=algoritms.R_TestIM);
	resetAndDisable(alg:=algoritms.S_AutoAVOM);
	resetAndDisable(alg:=algoritms.S_AutoTEN);
	resetAndDisable(alg:=algoritms.S_Test_IM);
	resetAndDisable(alg:=algoritms.S_Vibr);
	resetAndDisable(alg:=algoritms.S_Pms);
	resetAndDisable(alg:=algoritms.S_dPmg);
	resetAndDisable(alg:=algoritms.S_K);
	algoritms.S_I.CanRun:=FALSE;
	resetAndDisable(alg:=algoritms.S_V);
	resetAndDisable(alg:=algoritms.S_PP);
	resetAndDisable(alg:=algoritms.S_AP);
	algoritms.S_NO.CanRun:=TRUE;
	algoritms.S_AO.CanRun:=TRUE;
	resetAndDisable(alg:=algoritms.Test_IM);
	resetAndDisable(alg:=algoritms.Start_Test_P);
		resetAndDisable(alg:=algoritms.Test_P);
MODE_O:
	resetAndDisable(alg:=algoritms.Auto_Avom_);
	resetAndDisable(alg:=algoritms.autoNu_1);
	resetAndDisable(alg:=algoritms.autoNu_2);
	resetAndDisable(alg:=algoritms.autoPns);
	resetAndDisable(alg:=algoritms.AUto_Ten_);
	resetAndDisable(alg:=algoritms.PNS_ON_MV_);
	resetAndDisable(alg:=algoritms.no);
		resetAndDisable(alg:=algoritms.ao);
	resetAndDisable(alg:=algoritms.S_I);
	resetAndDisable(alg:=algoritms.Pms);
	resetAndDisable(alg:=algoritms.dPmg);
	resetAndDisable(alg:=algoritms.ppu);
	resetAndDisable(alg:=algoritms.F1_1);
	resetAndDisable(alg:=algoritms.F1_2);
	resetAndDisable(alg:=algoritms.F2_Ch);
	resetAndDisable(alg:=algoritms.F2_R);
	resetAndDisable(alg:=algoritms.F3);
	resetAndDisable(alg:=algoritms.F4);
	resetAndDisable(alg:=algoritms.Kr6_Move);
	resetAndDisable(alg:=algoritms.AutoPNS_Start);
	resetAndDisable(alg:=algoritms.R_AutoAVom);
	resetAndDisable(alg:=algoritms.R_AutoTEN);
	resetAndDisable(alg:=algoritms.R_TestIM);
	resetAndDisable(alg:=algoritms.S_AutoAVOM);
	resetAndDisable(alg:=algoritms.S_AutoTEN);
	resetAndDisable(alg:=algoritms.S_Test_IM);
	resetAndDisable(alg:=algoritms.S_Vibr);
	resetAndDisable(alg:=algoritms.S_Pms);
	resetAndDisable(alg:=algoritms.S_dPmg);
	resetAndDisable(alg:=algoritms.S_K);
	algoritms.Opres.CanRun:=FALSE;
	resetAndDisable(alg:=algoritms.S_V);
	resetAndDisable(alg:=algoritms.S_PP);
	resetAndDisable(alg:=algoritms.S_AP);
	algoritms.S_NO.CanRun:=TRUE;
	algoritms.S_AO.CanRun:=TRUE;
	resetAndDisable(alg:=algoritms.Test_IM);
	resetAndDisable(alg:=algoritms.Start_Test_P);
		resetAndDisable(alg:=algoritms.Test_P);
		
TEST_PROTECTIONS:	
		resetAndDisable(alg:=algoritms.Auto_Avom_);
		resetAndDisable(alg:=algoritms.autoNu_1);
		resetAndDisable(alg:=algoritms.autoNu_2);
		resetAndDisable(alg:=algoritms.autoPns);
		resetAndDisable(alg:=algoritms.AUto_Ten_);
		resetAndDisable(alg:=algoritms.PNS_ON_MV_);
		algoritms.no.CanRun:=TRUE;
		algoritms.ao.CanRun:=TRUE;
		resetAndDisable(alg:=algoritms.Opres);
		resetAndDisable(alg:=algoritms.Pms);
		resetAndDisable(alg:=algoritms.dPmg);
		resetAndDisable(alg:=algoritms.ppu);
		resetAndDisable(alg:=algoritms.F1_1);
		resetAndDisable(alg:=algoritms.F1_2);
		resetAndDisable(alg:=algoritms.F2_Ch);
		resetAndDisable(alg:=algoritms.F2_R);
		resetAndDisable(alg:=algoritms.F3);
		resetAndDisable(alg:=algoritms.F4);
		resetAndDisable(alg:=algoritms.Kr6_Move);
		resetAndDisable(alg:=algoritms.AutoPNS_Start);
		resetAndDisable(alg:=algoritms.R_AutoAVom);
		resetAndDisable(alg:=algoritms.R_AutoTEN);
		resetAndDisable(alg:=algoritms.R_TestIM);
		resetAndDisable(alg:=algoritms.S_AutoAVOM);
		resetAndDisable(alg:=algoritms.S_AutoTEN);
		resetAndDisable(alg:=algoritms.S_Test_IM);
		resetAndDisable(alg:=algoritms.S_Vibr);
		resetAndDisable(alg:=algoritms.S_dPmg);
		resetAndDisable(alg:=algoritms.S_I);
		resetAndDisable(alg:=algoritms.S_K);
		resetAndDisable(alg:=algoritms.S_Pms);
		resetAndDisable(alg:=algoritms.S_V);
		resetAndDisable(alg:=algoritms.S_AP);
		resetAndDisable(alg:=algoritms.S_PP);
		algoritms.S_NO.CanRun:=TRUE;
		algoritms.S_AO.CanRun:=TRUE;
		resetAndDisable(alg:=algoritms.Test_IM);
		Reset_ALL_P ();
		resetAndDisable(alg:=algoritms.Start_Test_P);
		algoritms.Test_P.CanRun:=TRUE;
		algoritms.Test_P.EnableOpcControl();

END_CASE

END_IF
END_METHOD

METHOD Public resetAndDisable
VAR_INPUT
	alg:REFERENCE TO BaseAlgoritm;
END_VAR
IF __ISVALIDREF(alg) THEN
	IF alg.isRuning THEN
		alg.reset();
	END_IF
	alg.CanRun:=FALSE;
END_IF
END_METHOD

END_FUNCTION_BLOCK

// K2/std12k5/AlgoritmsManager
	{attribute 'symbol' := 'none'}
FUNCTION_BLOCK AlgoritmsManager EXTENDS BaseAlgoritmsManager
VAR_INPUT
END_VAR
VAR_OUTPUT
	{attribute 'symbol' := 'read'}
	mode:ModeGpa;
	reg_V:BOOL;
END_VAR
VAR
	AoTrig:F_TRIG;
END_VAR

SUPER^();

METHOD PROTECTED onStart
VAR_INPUT
END_VAR
algoritms.opcComands.CanRun:=TRUE;
algoritms.opcComands.run();
///*ТЕМПЕРАТУРЫ*///////
(*Температуры т.1 - т.10*) 
		protections.p_TOpornogoPodshipnikaEDT_1.run();
		protections.p_TOpornoYpornogoPodshipnikaEDT_2.run();
		protections.p_TOpornoYpornogoPodshipnikaKolesaRedEDT_3.run();
		protections.p_TOpornoYpornogoPodshipnikaKolesaRedHT_4.run();
		protections.p_TOpornogoPodshipnikaShesterniReduktoraT_5.run();
		protections.p_TOpornogoPodshipnikaReduktoraHT_6.run();
		protections.p_TOpornoYpornogoPodshipnikaNagnetateljaT_7.run();
																										
		protections.p_TOpornoYpornogoPodshipnikaSvobodnogoKoncaNT_8.run();
		protections.p_TYpornogoPodshipnikaRavKolodokHT_9.run();
		protections.p_TYpornogoPodshipnikaNerabKolodokHT_10.run();
		protections.p_TgazaNaVyhodeH.run();
		
	(*Давления*)
		
		protections.p_OsSdvigNagnetatelja_Plus.run();
		protections.p_OsSdvigNagnetatelja_Minus.run();
		
	
	(*Дискретные сигналы *)
		
		
		protections.p_AO_PRU.run();
		protections.p_AO_fromSHU.run();
					
		algoritms.Synch_Rejim_.CanRun:=TRUE;
		algoritms.Synch_Rejim_.run ();
	
im.mv.DisableOpcControl ();
im.kran1.DisableOpcControl ();
im.kran2.DisableOpcControl ();
im.kran3.DisableOpcControl ();
im.kran3b.DisableOpcControl ();
im.kran4.DisableOpcControl ();
im.kran5.DisableOpcControl ();
END_METHOD

METHOD PROTECTED onInit
VAR_INPUT
END_VAR
VAR
	curObject:POINTER TO BaseObject;
	IcurAlg:AlgoritmInterface;
END_VAR
SUPER^.onInit();
setMode(nMode:=ModeGpa.MODE_STOP);
END_METHOD

METHOD PUBLIC setMode
VAR_INPUT
	nMode:ModeGpa;
END_VAR
IF 	nMode<>mode THEN
	mode:=nMode;
	CASE 	mode OF
	mode_stop:	resetAndDisable(alg:=algoritms.Auto_Avom_);
		resetAndDisable(alg:=algoritms.autoNu_1);
		resetAndDisable(alg:=algoritms.autoNu_2);
		resetAndDisable(alg:=algoritms.autoPns);
		resetAndDisable(alg:=algoritms.AUto_Ten_);
		resetAndDisable(alg:=algoritms.PNS_ON_MV_);
		resetAndDisable(alg:=algoritms.no);
		resetAndDisable(alg:=algoritms.ao);
		resetAndDisable(alg:=algoritms.Pms);
		resetAndDisable(alg:=algoritms.dPmg);
		resetAndDisable(alg:=algoritms.F1_1);
		resetAndDisable(alg:=algoritms.F1_2);
		resetAndDisable(alg:=algoritms.F2_Ch);
		resetAndDisable(alg:=algoritms.F2_R);
		resetAndDisable(alg:=algoritms.F3);
		resetAndDisable(alg:=algoritms.F4);
		resetAndDisable(alg:=algoritms.Kr6_Move);
		resetAndDisable(alg:=algoritms.AutoPNS_Start);
		resetAndDisable(alg:=algoritms.R_AutoAVom);
		resetAndDisable(alg:=algoritms.S_AutoAVOM);
		resetAndDisable(alg:=algoritms.S_Vibr);
		resetAndDisable(alg:=algoritms.S_dPmg);
		resetAndDisable(alg:=algoritms.S_I);
		resetAndDisable(alg:=algoritms.S_K);
		resetAndDisable(alg:=algoritms.S_Pms);
		resetAndDisable(alg:=algoritms.S_V);
		resetAndDisable(alg:=algoritms.S_AP);
		resetAndDisable(alg:=algoritms.S_PP);
		resetAndDisable(alg:=algoritms.Test_IM);
		algoritms.Opres.CanRun:=TRUE;
		algoritms.ppu.CanRun:=TRUE;
		resetAndDisable(alg:=algoritms.R_AutoTEN);
		//algoritms.R_AutoTEN.CanRun:=TRUE;
		algoritms.S_AutoTEN.CanRun:=TRUE;
		algoritms.S_Test_IM.CanRun:=TRUE;
		resetAndDisable(alg:=algoritms.R_TestIM);
		algoritms.S_NO.CanRun:=TRUE;
		algoritms.S_AO.CanRun:=TRUE;
		algmanager.reg_V:=FALSE;
		algoritms.Start_Test_P.CanRun:=TRUE;
		resetAndDisable(alg:=algoritms.Test_P);
		algoritms.Test_P.DisableOpcControl();
		
		////////////*АЛГОРИТМЫ РАБОТАЮЩИЕ В РЕЖИМЕ АВТОМАТИЧЕСКИЙ Реакторный  ПУСК*/////////////////////////////////
MODE_PUSKAP_R:
	resetAndDisable(alg:=algoritms.Auto_Avom_);
	resetAndDisable(alg:=algoritms.autoNu_1);
	resetAndDisable(alg:=algoritms.autoNu_2);
	resetAndDisable(alg:=algoritms.autoPns);
	resetAndDisable(alg:=algoritms.AUto_Ten_);
	resetAndDisable(alg:=algoritms.PNS_ON_MV_);
	resetAndDisable(alg:=algoritms.no);
	resetAndDisable(alg:=algoritms.ao);
	resetAndDisable(alg:=algoritms.Opres);
	resetAndDisable(alg:=algoritms.Pms);
	resetAndDisable(alg:=algoritms.dPmg);
	algoritms.ppu.CanRun:=TRUE;
	algoritms.ppu.run();
	resetAndDisable(alg:=algoritms.F1_2);
	resetAndDisable(alg:=algoritms.F2_Ch);
	resetAndDisable(alg:=algoritms.F2_R);
	resetAndDisable(alg:=algoritms.F3);
	resetAndDisable(alg:=algoritms.F4);
	resetAndDisable(alg:=algoritms.Kr6_Move);
	resetAndDisable(alg:=algoritms.AutoPNS_Start);
	resetAndDisable(alg:=algoritms.R_AutoAVom);
	resetAndDisable(alg:=algoritms.R_AutoTEN);
	resetAndDisable(alg:=algoritms.R_TestIM);
	resetAndDisable(alg:=algoritms.S_AutoAVOM);
	resetAndDisable(alg:=algoritms.S_AutoTEN);
	resetAndDisable(alg:=algoritms.S_Test_IM);
	resetAndDisable(alg:=algoritms.S_Vibr);
	resetAndDisable(alg:=algoritms.S_dPmg);
	resetAndDisable(alg:=algoritms.S_I);
	resetAndDisable(alg:=algoritms.S_K);
	resetAndDisable(alg:=algoritms.S_Pms);
	resetAndDisable(alg:=algoritms.S_V);
	resetAndDisable(alg:=algoritms.S_PP);
	algoritms.S_AP.CanRun:=FALSE;
	algoritms.S_NO.CanRun:=TRUE;
	algoritms.S_AO.CanRun:=TRUE;
	resetAndDisable(alg:=algoritms.Test_IM);
	resetAndDisable(alg:=algoritms.Start_Test_P);
	resetAndDisable(alg:=algoritms.Test_P);
MODE_PUSKAP_Ch:
	resetAndDisable(alg:=algoritms.Auto_Avom_);
	resetAndDisable(alg:=algoritms.autoNu_1);
	resetAndDisable(alg:=algoritms.autoNu_2);
	resetAndDisable(alg:=algoritms.autoPns);
	resetAndDisable(alg:=algoritms.AUto_Ten_);
	resetAndDisable(alg:=algoritms.PNS_ON_MV_);
	resetAndDisable(alg:=algoritms.no);
	resetAndDisable(alg:=algoritms.ao);
	resetAndDisable(alg:=algoritms.Opres);
	resetAndDisable(alg:=algoritms.Pms);
	resetAndDisable(alg:=algoritms.dPmg);
	algoritms.ppu.CanRun:=TRUE;
	algoritms.ppu.run();
	resetAndDisable(alg:=algoritms.F1_2);
	resetAndDisable(alg:=algoritms.F2_Ch);
	resetAndDisable(alg:=algoritms.F2_R);
	resetAndDisable(alg:=algoritms.F3);
	resetAndDisable(alg:=algoritms.F4);
	resetAndDisable(alg:=algoritms.Kr6_Move);
	resetAndDisable(alg:=algoritms.AutoPNS_Start);
	resetAndDisable(alg:=algoritms.R_AutoAVom);
	resetAndDisable(alg:=algoritms.R_AutoTEN);
	resetAndDisable(alg:=algoritms.R_TestIM);
	resetAndDisable(alg:=algoritms.S_AutoAVOM);
	resetAndDisable(alg:=algoritms.S_AutoTEN);
	resetAndDisable(alg:=algoritms.S_Test_IM);
	resetAndDisable(alg:=algoritms.S_Vibr);
	resetAndDisable(alg:=algoritms.S_dPmg);
	resetAndDisable(alg:=algoritms.S_I);
	resetAndDisable(alg:=algoritms.S_K);
	resetAndDisable(alg:=algoritms.S_Pms);
	resetAndDisable(alg:=algoritms.S_V);
	resetAndDisable(alg:=algoritms.S_PP);
	algoritms.S_AP.CanRun:=FALSE;
	algoritms.S_NO.CanRun:=TRUE;
	algoritms.S_AO.CanRun:=TRUE;
	resetAndDisable(alg:=algoritms.Test_IM);
	resetAndDisable(alg:=algoritms.Start_Test_P);
	resetAndDisable(alg:=algoritms.Test_P);
MODE_PUSKPP_R:
	resetAndDisable(alg:=algoritms.Auto_Avom_);
	resetAndDisable(alg:=algoritms.autoNu_1);
	resetAndDisable(alg:=algoritms.autoNu_2);
	resetAndDisable(alg:=algoritms.autoPns);
	resetAndDisable(alg:=algoritms.AUto_Ten_);
	resetAndDisable(alg:=algoritms.PNS_ON_MV_);
	resetAndDisable(alg:=algoritms.no);
	resetAndDisable(alg:=algoritms.ao);
	resetAndDisable(alg:=algoritms.Opres);
	resetAndDisable(alg:=algoritms.Pms);
	resetAndDisable(alg:=algoritms.dPmg);
	algoritms.ppu.CanRun:=TRUE;
	algoritms.ppu.run();
	resetAndDisable(alg:=algoritms.F1_2);
	resetAndDisable(alg:=algoritms.F2_Ch);
	resetAndDisable(alg:=algoritms.F2_R);
	resetAndDisable(alg:=algoritms.F3);
	resetAndDisable(alg:=algoritms.F4);
	resetAndDisable(alg:=algoritms.Kr6_Move);
	resetAndDisable(alg:=algoritms.AutoPNS_Start);
	resetAndDisable(alg:=algoritms.R_AutoAVom);
	resetAndDisable(alg:=algoritms.R_AutoTEN);
	resetAndDisable(alg:=algoritms.R_TestIM);
	resetAndDisable(alg:=algoritms.S_AutoAVOM);
	resetAndDisable(alg:=algoritms.S_AutoTEN);
	resetAndDisable(alg:=algoritms.S_Test_IM);
	resetAndDisable(alg:=algoritms.S_Vibr);
	resetAndDisable(alg:=algoritms.S_dPmg);
	resetAndDisable(alg:=algoritms.S_I);
	resetAndDisable(alg:=algoritms.S_K);
	resetAndDisable(alg:=algoritms.S_Pms);
	resetAndDisable(alg:=algoritms.S_V);
	resetAndDisable(alg:=algoritms.S_AP);
	algoritms.S_PP.CanRun:=FALSE;
	algoritms.S_NO.CanRun:=TRUE;
	algoritms.S_AO.CanRun:=TRUE;
	resetAndDisable(alg:=algoritms.Test_IM);
	resetAndDisable(alg:=algoritms.Start_Test_P);
	resetAndDisable(alg:=algoritms.Test_P);
MODE_PUSKPP_Ch:
	resetAndDisable(alg:=algoritms.Auto_Avom_);
	resetAndDisable(alg:=algoritms.autoNu_1);
	resetAndDisable(alg:=algoritms.autoNu_2);
	resetAndDisable(alg:=algoritms.autoPns);
	resetAndDisable(alg:=algoritms.AUto_Ten_);
	resetAndDisable(alg:=algoritms.PNS_ON_MV_);
	resetAndDisable(alg:=algoritms.no);
	resetAndDisable(alg:=algoritms.ao);
	resetAndDisable(alg:=algoritms.Opres);
	resetAndDisable(alg:=algoritms.Pms);
	resetAndDisable(alg:=algoritms.dPmg);
	algoritms.ppu.CanRun:=TRUE;
	algoritms.ppu.run();
	resetAndDisable(alg:=algoritms.F1_2);
	resetAndDisable(alg:=algoritms.F2_Ch);
	resetAndDisable(alg:=algoritms.F2_R);
	resetAndDisable(alg:=algoritms.F3);
	resetAndDisable(alg:=algoritms.F4);
	resetAndDisable(alg:=algoritms.Kr6_Move);
	resetAndDisable(alg:=algoritms.AutoPNS_Start);
	resetAndDisable(alg:=algoritms.R_AutoAVom);
	resetAndDisable(alg:=algoritms.R_AutoTEN);
	resetAndDisable(alg:=algoritms.R_TestIM);
	resetAndDisable(alg:=algoritms.S_AutoAVOM);
	resetAndDisable(alg:=algoritms.S_AutoTEN);
	resetAndDisable(alg:=algoritms.S_Test_IM);
	resetAndDisable(alg:=algoritms.S_Vibr);
	resetAndDisable(alg:=algoritms.S_dPmg);
	resetAndDisable(alg:=algoritms.S_I);
	resetAndDisable(alg:=algoritms.S_K);
	resetAndDisable(alg:=algoritms.S_Pms);
	resetAndDisable(alg:=algoritms.S_V);
	resetAndDisable(alg:=algoritms.S_AP);
	algoritms.S_PP.CanRun:=FALSE;
	algoritms.S_NO.CanRun:=TRUE;
	algoritms.S_AO.CanRun:=TRUE;
	resetAndDisable(alg:=algoritms.Test_IM);
	resetAndDisable(alg:=algoritms.Start_Test_P);
	resetAndDisable(alg:=algoritms.Test_P);
MODE_WORK_M:
	resetAndDisable(alg:=algoritms.autoNu_1);
	resetAndDisable(alg:=algoritms.AUto_Ten_);
	resetAndDisable(alg:=algoritms.PNS_ON_MV_);
	resetAndDisable(alg:=algoritms.no);
	resetAndDisable(alg:=algoritms.ao);
	resetAndDisable(alg:=algoritms.Opres);
	resetAndDisable(alg:=algoritms.Pms);
	resetAndDisable(alg:=algoritms.dPmg);
	algoritms.ppu.CanRun:=TRUE;
	algoritms.ppu.run();
	resetAndDisable(alg:=algoritms.F1_1);
	resetAndDisable(alg:=algoritms.F1_2);
	resetAndDisable(alg:=algoritms.F2_Ch);
	resetAndDisable(alg:=algoritms.F2_R);
	resetAndDisable(alg:=algoritms.F3);
	resetAndDisable(alg:=algoritms.F4);
	resetAndDisable(alg:=algoritms.R_AutoTEN);
	resetAndDisable(alg:=algoritms.R_TestIM);
	resetAndDisable(alg:=algoritms.S_AutoTEN);
	resetAndDisable(alg:=algoritms.S_Test_IM);
	resetAndDisable(alg:=algoritms.S_dPmg);
	resetAndDisable(alg:=algoritms.S_I);
	resetAndDisable(alg:=algoritms.S_K);
	resetAndDisable(alg:=algoritms.S_Pms);
	resetAndDisable(alg:=algoritms.S_V);
	resetAndDisable(alg:=algoritms.S_AP);
	resetAndDisable(alg:=algoritms.S_PP);
	algoritms.S_NO.CanRun:=TRUE;
	algoritms.S_AO.CanRun:=TRUE;
	resetAndDisable(alg:=algoritms.Test_IM);
	resetAndDisable(alg:=algoritms.Start_Test_P);
	resetAndDisable(alg:=algoritms.Test_P);
MODE_WORK_K:
	resetAndDisable(alg:=algoritms.autoNu_1);
	resetAndDisable(alg:=algoritms.AUto_Ten_);
	resetAndDisable(alg:=algoritms.PNS_ON_MV_);
	resetAndDisable(alg:=algoritms.no);
	resetAndDisable(alg:=algoritms.ao);
	resetAndDisable(alg:=algoritms.Opres);
	resetAndDisable(alg:=algoritms.Pms);
	resetAndDisable(alg:=algoritms.dPmg);
	algoritms.ppu.CanRun:=TRUE;
	algoritms.ppu.run();
	resetAndDisable(alg:=algoritms.F1_1);
	resetAndDisable(alg:=algoritms.F1_2);
	resetAndDisable(alg:=algoritms.F2_Ch);
	resetAndDisable(alg:=algoritms.F2_R);
	resetAndDisable(alg:=algoritms.F3);
	resetAndDisable(alg:=algoritms.F4);
	resetAndDisable(alg:=algoritms.R_AutoTEN);
	resetAndDisable(alg:=algoritms.R_TestIM);
	resetAndDisable(alg:=algoritms.S_AutoTEN);
	resetAndDisable(alg:=algoritms.S_Test_IM);
	resetAndDisable(alg:=algoritms.S_dPmg);
	resetAndDisable(alg:=algoritms.S_I);
	resetAndDisable(alg:=algoritms.S_K);
	resetAndDisable(alg:=algoritms.S_Pms);
	resetAndDisable(alg:=algoritms.S_V);
	resetAndDisable(alg:=algoritms.S_AP);
	resetAndDisable(alg:=algoritms.S_PP);
	algoritms.S_NO.CanRun:=TRUE;
	algoritms.S_AO.CanRun:=TRUE;
	resetAndDisable(alg:=algoritms.Test_IM);
	resetAndDisable(alg:=algoritms.Start_Test_P);
	resetAndDisable(alg:=algoritms.Test_P);
MODE_NO:
		resetAndDisable(alg:=algoritms.AUto_Ten_);
		resetAndDisable(alg:=algoritms.PNS_ON_MV_);
		resetAndDisable(alg:=algoritms.ao);
		resetAndDisable(alg:=algoritms.Opres);
		resetAndDisable(alg:=algoritms.Pms);
		resetAndDisable(alg:=algoritms.dPmg);
		resetAndDisable(alg:=algoritms.ppu);
		resetAndDisable(alg:=algoritms.F1_1);
		resetAndDisable(alg:=algoritms.F1_2);
		resetAndDisable(alg:=algoritms.F2_Ch);
		resetAndDisable(alg:=algoritms.F2_R);
		resetAndDisable(alg:=algoritms.F3);
		resetAndDisable(alg:=algoritms.F4);
		resetAndDisable(alg:=algoritms.Kr6_Move);
		resetAndDisable(alg:=algoritms.AutoPNS_Start);
		//resetAndDisable(alg:=algoritms.R_AutoAVom);
		resetAndDisable(alg:=algoritms.R_AutoTEN);
		resetAndDisable(alg:=algoritms.R_TestIM);
		//resetAndDisable(alg:=algoritms.S_AutoAVOM);
		resetAndDisable(alg:=algoritms.S_AutoTEN);
		resetAndDisable(alg:=algoritms.S_Test_IM);
		resetAndDisable(alg:=algoritms.S_dPmg);
		resetAndDisable(alg:=algoritms.S_I);
		resetAndDisable(alg:=algoritms.S_K);
		resetAndDisable(alg:=algoritms.S_Pms);
		resetAndDisable(alg:=algoritms.S_V);
		resetAndDisable(alg:=algoritms.S_AP);
		resetAndDisable(alg:=algoritms.S_PP);
		resetAndDisable(alg:=algoritms.S_NO);
		algoritms.S_AO.CanRun:=TRUE;
		resetAndDisable(alg:=algoritms.Test_IM);
		resetAndDisable(alg:=algoritms.Start_Test_P);
	resetAndDisable(alg:=algoritms.Test_P);
MODE_AO:
		resetAndDisable(alg:=algoritms.AUto_Ten_);
		resetAndDisable(alg:=algoritms.PNS_ON_MV_);
		resetAndDisable(alg:=algoritms.no);
		resetAndDisable(alg:=algoritms.Opres);
		resetAndDisable(alg:=algoritms.Pms);
		resetAndDisable(alg:=algoritms.dPmg);
		resetAndDisable(alg:=algoritms.ppu);
		resetAndDisable(alg:=algoritms.F1_1);
		resetAndDisable(alg:=algoritms.F1_2);
		resetAndDisable(alg:=algoritms.F2_Ch);
		resetAndDisable(alg:=algoritms.F2_R);
		resetAndDisable(alg:=algoritms.F3);
		resetAndDisable(alg:=algoritms.F4);
		resetAndDisable(alg:=algoritms.Kr6_Move);
		resetAndDisable(alg:=algoritms.AutoPNS_Start);
		//resetAndDisable(alg:=algoritms.R_AutoAVom);
		resetAndDisable(alg:=algoritms.R_AutoTEN);
		resetAndDisable(alg:=algoritms.R_TestIM);
		//resetAndDisable(alg:=algoritms.S_AutoAVOM);
		resetAndDisable(alg:=algoritms.S_AutoTEN);
		resetAndDisable(alg:=algoritms.S_Test_IM);
		resetAndDisable(alg:=algoritms.S_dPmg);
		resetAndDisable(alg:=algoritms.S_I);
		resetAndDisable(alg:=algoritms.S_K);
		resetAndDisable(alg:=algoritms.S_Pms);
		resetAndDisable(alg:=algoritms.S_V);
		resetAndDisable(alg:=algoritms.S_AP);
		resetAndDisable(alg:=algoritms.S_PP);
		resetAndDisable(alg:=algoritms.S_NO);
		resetAndDisable(alg:=algoritms.S_AO);
		resetAndDisable(alg:=algoritms.Test_IM);
		resetAndDisable(alg:=algoritms.Start_Test_P);
	resetAndDisable(alg:=algoritms.Test_P);
MODE_EO:		
		resetAndDisable(alg:=algoritms.Auto_Avom_);
		resetAndDisable(alg:=algoritms.autoNu_1);
		resetAndDisable(alg:=algoritms.autoNu_2);
		resetAndDisable(alg:=algoritms.autoPns);
		resetAndDisable(alg:=algoritms.AUto_Ten_);
		resetAndDisable(alg:=algoritms.PNS_ON_MV_);
		resetAndDisable(alg:=algoritms.no);
		resetAndDisable(alg:=algoritms.ao);
		resetAndDisable(alg:=algoritms.Opres);
		resetAndDisable(alg:=algoritms.Pms);
		resetAndDisable(alg:=algoritms.dPmg);
		resetAndDisable(alg:=algoritms.ppu);
		resetAndDisable(alg:=algoritms.F1_1);
		resetAndDisable(alg:=algoritms.F1_2);
		resetAndDisable(alg:=algoritms.F2_Ch);
		resetAndDisable(alg:=algoritms.F2_R);
		resetAndDisable(alg:=algoritms.F3);
		resetAndDisable(alg:=algoritms.F4);
		resetAndDisable(alg:=algoritms.Kr6_Move);
		resetAndDisable(alg:=algoritms.AutoPNS_Start);
		resetAndDisable(alg:=algoritms.R_AutoAVom);
		resetAndDisable(alg:=algoritms.R_AutoTEN);
		resetAndDisable(alg:=algoritms.R_TestIM);
		resetAndDisable(alg:=algoritms.S_AutoAVOM);
		resetAndDisable(alg:=algoritms.S_AutoTEN);
		resetAndDisable(alg:=algoritms.S_Test_IM);
		resetAndDisable(alg:=algoritms.S_Vibr);
		resetAndDisable(alg:=algoritms.S_dPmg);
		resetAndDisable(alg:=algoritms.S_I);
		resetAndDisable(alg:=algoritms.S_K);
		resetAndDisable(alg:=algoritms.S_Pms);
		resetAndDisable(alg:=algoritms.S_V);
		resetAndDisable(alg:=algoritms.S_AP);
		resetAndDisable(alg:=algoritms.S_PP);
		resetAndDisable(alg:=algoritms.S_NO);
		resetAndDisable(alg:=algoritms.S_AO);
		resetAndDisable(alg:=algoritms.Test_IM);
		Reset_ALL_P ();
		resetAndDisable(alg:=algoritms.Start_Test_P);
	resetAndDisable(alg:=algoritms.Test_P);

